LIN {X 0,Y 581.14,Z 534.428,A -85,B 0,C 180,E1 -1994.848,E2 -1994.848} C_VEL
LIN {X 0,Y 580.577,Z 528.636,A -85,B 0,C 180,E1 -1994.951,E2 -1994.951} C_VEL
LIN {X 0,Y 575.005,Z 509.982,A -85,B 0,C 180,E1 -1995.336,E2 -1995.336} C_VEL
LIN {X 0,Y 574.391,Z 504.171,A -85,B 0,C 180,E1 -1995.426,E2 -1995.426} C_VEL
LIN {X 0,Y 574.468,Z 402.044,A -85,B 0,C 180,E1 -1996.725,E2 -1996.725} C_VEL
LIN {X 0,Y 573.703,Z 397.536,A -85,B 0,C 180,E1 -1996.823,E2 -1996.823} C_VEL
LIN {X 0,Y 573.883,Z 376.717,A -85,B 0,C 180,E1 -1999.443,E2 -1999.443} C_VEL
LIN {X 0,Y 574.185,Z 354.585,A -85,B 0,C 180,E1 -2002.299,E2 -2002.299} C_VEL
LIN {X 0,Y 574.353,Z 340.111,A -85,B 0,C 180,E1 -2004.2,E2 -2004.2} C_VEL
LIN {X 0,Y 573.485,Z 334.982,A -85,B 0,C 180,E1 -2004.924,E2 -2004.924} C_VEL
LIN {X 0,Y 573.218,Z 333.802,A -85,B 0,C 180,E1 -2005.15,E2 -2005.15} C_VEL
LIN {X 0,Y 573.188,Z 333.715,A -85,B 0,C 180,E1 -2008.016,E2 -2008.016} C_VEL
LIN {X 0,Y 573.207,Z 333.705,A -85,B 0,C 180,E1 -2010.878,E2 -2010.878} C_VEL
LIN {X 0,Y 573.216,Z 333.705,A -85,B 0,C 180,E1 -2013.517,E2 -2013.517} C_VEL
LIN {X 0,Y 573.178,Z 333.717,A -85,B 0,C 180,E1 -2016.054,E2 -2016.054} C_VEL
LIN {X 0,Y 573.212,Z 333.704,A -85,B 0,C 180,E1 -2018.704,E2 -2018.704} C_VEL
LIN {X 0,Y 573.184,Z 333.709,A -85,B 0,C 180,E1 -2021.587,E2 -2021.587} C_VEL
LIN {X 0,Y 573.203,Z 333.71,A -85,B 0,C 180,E1 -2024.337,E2 -2024.337} C_VEL
LIN {X 0,Y 573.207,Z 333.702,A -85,B 0,C 180,E1 -2027.362,E2 -2027.362} C_VEL
LIN {X 0,Y 573.219,Z 333.704,A -85,B 0,C 180,E1 -2030.572,E2 -2030.572} C_VEL
LIN {X 0,Y 573.199,Z 333.703,A -85,B 0,C 180,E1 -2033.073,E2 -2033.073} C_VEL
LIN {X 0,Y 573.237,Z 333.704,A -85,B 0,C 180,E1 -2035.669,E2 -2035.669} C_VEL
LIN {X 0,Y 573.207,Z 333.713,A -85,B 0,C 180,E1 -2038.182,E2 -2038.182} C_VEL
LIN {X 0,Y 573.218,Z 333.707,A -85,B 0,C 180,E1 -2040.631,E2 -2040.631} C_VEL
LIN {X 0,Y 573.235,Z 333.849,A -85,B 0,C 180,E1 -2042.826,E2 -2042.826} C_VEL
LIN {X 0,Y 574.862,Z 341.006,A -85,B 0,C 180,E1 -2043.754,E2 -2043.754} C_VEL
LIN {X 0,Y 574.556,Z 361.798,A -85,B 0,C 180,E1 -2046.193,E2 -2046.193} C_VEL
LIN {X 0,Y 574.194,Z 387.884,A -85,B 0,C 180,E1 -2049.209,E2 -2049.209} C_VEL
LIN {X 0,Y 574.072,Z 398.599,A -85,B 0,C 180,E1 -2050.415,E2 -2050.415} C_VEL
LIN {X 0,Y 575.202,Z 405.826,A -85,B 0,C 180,E1 -2050.567,E2 -2050.567} C_VEL
LIN {X 0,Y 574.722,Z 563.783,A -85,B 0,C 180,E1 -2052.608,E2 -2052.608} C_VEL
LIN {X 0,Y 574.651,Z 578.295,A -85,B 0,C 180,E1 -2052.915,E2 -2052.915} C_VEL
LIN {X 0,Y 574.422,Z 594.793,A -85,B 0,C 180,E1 -2053.428,E2 -2053.428} C_VEL
LIN {X 0,Y 574.286,Z 608.726,A -85,B 0,C 180,E1 -2054.017,E2 -2054.017} C_VEL
LIN {X 0,Y 574.055,Z 620.862,A -85,B 0,C 180,E1 -2054.648,E2 -2054.648} C_VEL
LIN {X 0,Y 573.885,Z 634.297,A -85,B 0,C 180,E1 -2055.496,E2 -2055.496} C_VEL
LIN {X 0,Y 573.651,Z 647.761,A -85,B 0,C 180,E1 -2056.539,E2 -2056.539} C_VEL
LIN {X 0,Y 573.524,Z 657.489,A -85,B 0,C 180,E1 -2057.437,E2 -2057.437} C_VEL
LIN {X 0,Y 573.349,Z 667.502,A -85,B 0,C 180,E1 -2058.51,E2 -2058.51} C_VEL
LIN {X 0,Y 573.274,Z 677.322,A -85,B 0,C 180,E1 -2059.76,E2 -2059.76} C_VEL
LIN {X 0,Y 573.133,Z 686.46,A -85,B 0,C 180,E1 -2061.183,E2 -2061.183} C_VEL
LIN {X 0,Y 573.095,Z 692.191,A -85,B 0,C 180,E1 -2062.247,E2 -2062.247} C_VEL
LIN {X 0,Y 573.013,Z 698.405,A -85,B 0,C 180,E1 -2063.662,E2 -2063.662} C_VEL
LIN {X 0,Y 572.998,Z 702.164,A -85,B 0,C 180,E1 -2064.722,E2 -2064.722} C_VEL
LIN {X 0,Y 573.008,Z 705.165,A -85,B 0,C 180,E1 -2065.78,E2 -2065.78} C_VEL
LIN {X 0,Y 572.953,Z 708.114,A -85,B 0,C 180,E1 -2067.188,E2 -2067.188} C_VEL
LIN {X 0,Y 572.942,Z 709.884,A -85,B 0,C 180,E1 -2068.594,E2 -2068.594} C_VEL
LIN {X 0,Y 572.936,Z 710.496,A -85,B 0,C 180,E1 -2070,E2 -2070} C_VEL
LIN {X 0,Y 572.944,Z 709.958,A -85,B 0,C 180,E1 -2071.406,E2 -2071.406} C_VEL
LIN {X 0,Y 572.956,Z 708.262,A -85,B 0,C 180,E1 -2072.812,E2 -2072.812} C_VEL
LIN {X 0,Y 573.008,Z 705.388,A -85,B 0,C 180,E1 -2074.22,E2 -2074.22} C_VEL
LIN {X 0,Y 573.054,Z 701.325,A -85,B 0,C 180,E1 -2075.63,E2 -2075.63} C_VEL
LIN {X 0,Y 573.049,Z 695.916,A -85,B 0,C 180,E1 -2077.045,E2 -2077.045} C_VEL
LIN {X 0,Y 573.099,Z 688.976,A -85,B 0,C 180,E1 -2078.462,E2 -2078.462} C_VEL
LIN {X 0,Y 573.188,Z 681.545,A -85,B 0,C 180,E1 -2079.706,E2 -2079.706} C_VEL
LIN {X 0,Y 573.287,Z 673.107,A -85,B 0,C 180,E1 -2080.89,E2 -2080.89} C_VEL
LIN {X 0,Y 573.406,Z 663.566,A -85,B 0,C 180,E1 -2082.026,E2 -2082.026} C_VEL
LIN {X 0,Y 573.609,Z 651.863,A -85,B 0,C 180,E1 -2083.191,E2 -2083.191} C_VEL
LIN {X 0,Y 573.777,Z 639.91,A -85,B 0,C 180,E1 -2084.18,E2 -2084.18} C_VEL
LIN {X 0,Y 574.002,Z 628.328,A -85,B 0,C 180,E1 -2084.99,E2 -2084.99} C_VEL
LIN {X 0,Y 574.168,Z 616.021,A -85,B 0,C 180,E1 -2085.713,E2 -2085.713} C_VEL
LIN {X 0,Y 574.347,Z 600.523,A -85,B 0,C 180,E1 -2086.437,E2 -2086.437} C_VEL
LIN {X 0,Y 574.505,Z 586.676,A -85,B 0,C 180,E1 -2086.936,E2 -2086.936} C_VEL
LIN {X 0,Y 574.677,Z 572.66,A -85,B 0,C 180,E1 -2087.311,E2 -2087.311} C_VEL
LIN {X 0,Y 574.793,Z 556.718,A -85,B 0,C 180,E1 -2087.589,E2 -2087.589} C_VEL
LIN {X 0,Y 575.167,Z 404.401,A -85,B 0,C 180,E1 -2089.542,E2 -2089.542} C_VEL
LIN {X 0,Y 574.062,Z 398.56,A -85,B 0,C 180,E1 -2089.678,E2 -2089.678} C_VEL
LIN {X 0,Y 574.415,Z 372.355,A -85,B 0,C 180,E1 -2092.669,E2 -2092.669} C_VEL
LIN {X 0,Y 574.801,Z 346.251,A -85,B 0,C 180,E1 -2095.725,E2 -2095.725} C_VEL
LIN {X 0,Y 574.791,Z 340.48,A -85,B 0,C 180,E1 -2096.4,E2 -2096.4} C_VEL
LIN {X 0,Y 573.231,Z 333.822,A -85,B 0,C 180,E1 -2097.273,E2 -2097.273} C_VEL
LIN {X 0,Y 573.219,Z 333.71,A -85,B 0,C 180,E1 -2100.178,E2 -2100.178} C_VEL
LIN {X 0,Y 573.216,Z 333.704,A -85,B 0,C 180,E1 -2102.647,E2 -2102.647} C_VEL
LIN {X 0,Y 573.178,Z 333.709,A -85,B 0,C 180,E1 -2105.19,E2 -2105.19} C_VEL
LIN {X 0,Y 573.207,Z 333.712,A -85,B 0,C 180,E1 -2107.81,E2 -2107.81} C_VEL
LIN {X 0,Y 573.199,Z 333.706,A -85,B 0,C 180,E1 -2110.529,E2 -2110.529} C_VEL
LIN {X 0,Y 573.193,Z 333.707,A -85,B 0,C 180,E1 -2113.363,E2 -2113.363} C_VEL
LIN {X 0,Y 573.217,Z 333.709,A -85,B 0,C 180,E1 -2115.665,E2 -2115.665} C_VEL
LIN {X 0,Y 573.191,Z 333.707,A -85,B 0,C 180,E1 -2118.539,E2 -2118.539} C_VEL
LIN {X 0,Y 573.229,Z 333.703,A -85,B 0,C 180,E1 -2121.297,E2 -2121.297} C_VEL
LIN {X 0,Y 573.184,Z 333.711,A -85,B 0,C 180,E1 -2124.023,E2 -2124.023} C_VEL
LIN {X 0,Y 573.231,Z 333.701,A -85,B 0,C 180,E1 -2126.515,E2 -2126.515} C_VEL
LIN {X 0,Y 573.224,Z 333.701,A -85,B 0,C 180,E1 -2129.119,E2 -2129.119} C_VEL
LIN {X 0,Y 573.219,Z 333.705,A -85,B 0,C 180,E1 -2131.977,E2 -2131.977} C_VEL
LIN {X 0,Y 573.223,Z 333.701,A -85,B 0,C 180,E1 -2134.588,E2 -2134.588} C_VEL
LIN {X 0,Y 573.236,Z 333.7,A -85,B 0,C 180,E1 -2136.901,E2 -2136.901} C_VEL
LIN {X 0,Y 573.249,Z 333.7,A -85,B 0,C 180,E1 -2139.173,E2 -2139.173} C_VEL
LIN {X 0,Y 573.21,Z 333.71,A -85,B 0,C 180,E1 -2141.411,E2 -2141.411} C_VEL
LIN {X 0,Y 573.238,Z 333.707,A -85,B 0,C 180,E1 -2143.621,E2 -2143.621} C_VEL
LIN {X 0,Y 573.272,Z 333.701,A -85,B 0,C 180,E1 -2145.807,E2 -2145.807} C_VEL
LIN {X 0,Y 573.265,Z 333.694,A -85,B 0,C 180,E1 -2148.745,E2 -2148.745} C_VEL
LIN {X 0,Y 573.281,Z 333.704,A -85,B 0,C 180,E1 -2151.54,E2 -2151.54} C_VEL
LIN {X 0,Y 573.244,Z 333.704,A -85,B 0,C 180,E1 -2153.665,E2 -2153.665} C_VEL
LIN {X 0,Y 573.228,Z 333.704,A -85,B 0,C 180,E1 -2155.781,E2 -2155.781} C_VEL
LIN {X 0,Y 573.314,Z 333.693,A -85,B 0,C 180,E1 -2157.892,E2 -2157.892} C_VEL
LIN {X 0,Y 573.32,Z 333.689,A -85,B 0,C 180,E1 -2160.702,E2 -2160.702} C_VEL
LIN {X 0,Y 573.294,Z 333.692,A -85,B 0,C 180,E1 -2162.811,E2 -2162.811} C_VEL
LIN {X 0,Y 573.295,Z 333.697,A -85,B 0,C 180,E1 -2165.628,E2 -2165.628} C_VEL
LIN {X 0,Y 573.255,Z 333.695,A -85,B 0,C 180,E1 -2168.46,E2 -2168.46} C_VEL
LIN {X 0,Y 573.274,Z 333.704,A -85,B 0,C 180,E1 -2171.312,E2 -2171.312} C_VEL
LIN {X 0,Y 573.261,Z 333.694,A -85,B 0,C 180,E1 -2174.193,E2 -2174.193} C_VEL
LIN {X 0,Y 573.259,Z 333.704,A -85,B 0,C 180,E1 -2177.111,E2 -2177.111} C_VEL
LIN {X 0,Y 573.241,Z 333.697,A -85,B 0,C 180,E1 -2180.077,E2 -2180.077} C_VEL
LIN {X 0,Y 573.235,Z 333.7,A -85,B 0,C 180,E1 -2182.338,E2 -2182.338} C_VEL
LIN {X 0,Y 573.254,Z 333.703,A -85,B 0,C 180,E1 -2185.41,E2 -2185.41} C_VEL
LIN {X 0,Y 573.25,Z 333.698,A -85,B 0,C 180,E1 -2188.029,E2 -2188.029} C_VEL
LIN {X 0,Y 573.234,Z 333.704,A -85,B 0,C 180,E1 -2190.883,E2 -2190.883} C_VEL
LIN {X 0,Y 573.263,Z 333.698,A -85,B 0,C 180,E1 -2193.524,E2 -2193.524} C_VEL
LIN {X 0,Y 573.215,Z 333.702,A -85,B 0,C 180,E1 -2196.051,E2 -2196.051} C_VEL
LIN {X 0,Y 573.25,Z 333.701,A -85,B 0,C 180,E1 -2198.701,E2 -2198.701} C_VEL
LIN {X 0,Y 573.244,Z 333.699,A -85,B 0,C 180,E1 -2201.594,E2 -2201.594} C_VEL
LIN {X 0,Y 573.236,Z 333.701,A -85,B 0,C 180,E1 -2204.333,E2 -2204.333} C_VEL
LIN {X 0,Y 573.24,Z 333.702,A -85,B 0,C 180,E1 -2207.358,E2 -2207.358} C_VEL
LIN {X 0,Y 573.248,Z 333.701,A -85,B 0,C 180,E1 -2210.393,E2 -2210.393} C_VEL
LIN {X 0,Y 573.253,Z 333.705,A -85,B 0,C 180,E1 -2213.078,E2 -2213.078} C_VEL
LIN {X 0,Y 573.266,Z 333.697,A -85,B 0,C 180,E1 -2215.671,E2 -2215.671} C_VEL
LIN {X 0,Y 573.247,Z 333.7,A -85,B 0,C 180,E1 -2218.185,E2 -2218.185} C_VEL
LIN {X 0,Y 573.264,Z 333.704,A -85,B 0,C 180,E1 -2220.634,E2 -2220.634} C_VEL
LIN {X 0,Y 573.273,Z 333.826,A -85,B 0,C 180,E1 -2223.522,E2 -2223.522} C_VEL
LIN {X 0,Y 574.8,Z 339.819,A -85,B 0,C 180,E1 -2224.275,E2 -2224.275} C_VEL
LIN {X 0,Y 574.832,Z 350.617,A -85,B 0,C 180,E1 -2225.437,E2 -2225.437} C_VEL
LIN {X 0,Y 574.354,Z 379.411,A -85,B 0,C 180,E1 -2228.464,E2 -2228.464} C_VEL
LIN {X 0,Y 574.163,Z 397.928,A -85,B 0,C 180,E1 -2230.363,E2 -2230.363} C_VEL
LIN {X 0,Y 575.245,Z 404.725,A -85,B 0,C 180,E1 -2230.51,E2 -2230.51} C_VEL
LIN {X 0,Y 574.744,Z 565.38,A -85,B 0,C 180,E1 -2232.586,E2 -2232.586} C_VEL
LIN {X 0,Y 574.616,Z 580.708,A -85,B 0,C 180,E1 -2232.93,E2 -2232.93} C_VEL
LIN {X 0,Y 574.433,Z 596.043,A -85,B 0,C 180,E1 -2233.428,E2 -2233.428} C_VEL
LIN {X 0,Y 574.292,Z 609.771,A -85,B 0,C 180,E1 -2234.017,E2 -2234.017} C_VEL
LIN {X 0,Y 574.032,Z 623.244,A -85,B 0,C 180,E1 -2234.738,E2 -2234.738} C_VEL
LIN {X 0,Y 573.861,Z 636.818,A -85,B 0,C 180,E1 -2235.632,E2 -2235.632} C_VEL
LIN {X 0,Y 573.635,Z 649.35,A -85,B 0,C 180,E1 -2236.629,E2 -2236.629} C_VEL
LIN {X 0,Y 573.477,Z 659.749,A -85,B 0,C 180,E1 -2237.616,E2 -2237.616} C_VEL
LIN {X 0,Y 573.286,Z 669.77,A -85,B 0,C 180,E1 -2238.734,E2 -2238.734} C_VEL
LIN {X 0,Y 573.243,Z 678.858,A -85,B 0,C 180,E1 -2239.939,E2 -2239.939} C_VEL
LIN {X 0,Y 573.132,Z 686.734,A -85,B 0,C 180,E1 -2241.183,E2 -2241.183} C_VEL
LIN {X 0,Y 573.074,Z 694.089,A -85,B 0,C 180,E1 -2242.602,E2 -2242.602} C_VEL
LIN {X 0,Y 573.041,Z 699.923,A -85,B 0,C 180,E1 -2244.016,E2 -2244.016} C_VEL
LIN {X 0,Y 572.951,Z 703.385,A -85,B 0,C 180,E1 -2245.074,E2 -2245.074} C_VEL
LIN {X 0,Y 573.005,Z 706.889,A -85,B 0,C 180,E1 -2246.484,E2 -2246.484} C_VEL
LIN {X 0,Y 572.938,Z 709.192,A -85,B 0,C 180,E1 -2247.891,E2 -2247.891} C_VEL
LIN {X 0,Y 572.936,Z 710.349,A -85,B 0,C 180,E1 -2249.297,E2 -2249.297} C_VEL
LIN {X 0,Y 572.936,Z 710.349,A -85,B 0,C 180,E1 -2250.703,E2 -2250.703} C_VEL
LIN {X 0,Y 572.938,Z 709.191,A -85,B 0,C 180,E1 -2252.109,E2 -2252.109} C_VEL
LIN {X 0,Y 573.005,Z 706.887,A -85,B 0,C 180,E1 -2253.516,E2 -2253.516} C_VEL
LIN {X 0,Y 572.951,Z 703.385,A -85,B 0,C 180,E1 -2254.926,E2 -2254.926} C_VEL
LIN {X 0,Y 573.013,Z 698.608,A -85,B 0,C 180,E1 -2256.338,E2 -2256.338} C_VEL
LIN {X 0,Y 573.094,Z 692.422,A -85,B 0,C 180,E1 -2257.753,E2 -2257.753} C_VEL
LIN {X 0,Y 573.135,Z 684.648,A -85,B 0,C 180,E1 -2259.173,E2 -2259.173} C_VEL
LIN {X 0,Y 573.27,Z 676.368,A -85,B 0,C 180,E1 -2260.418,E2 -2260.418} C_VEL
LIN {X 0,Y 573.386,Z 666.39,A -85,B 0,C 180,E1 -2261.668,E2 -2261.668} C_VEL
LIN {X 0,Y 573.568,Z 656.188,A -85,B 0,C 180,E1 -2262.742,E2 -2262.742} C_VEL
LIN {X 0,Y 573.705,Z 644.017,A -85,B 0,C 180,E1 -2263.82,E2 -2263.82} C_VEL
LIN {X 0,Y 573.962,Z 630.901,A -85,B 0,C 180,E1 -2264.781,E2 -2264.781} C_VEL
LIN {X 0,Y 574.141,Z 616.867,A -85,B 0,C 180,E1 -2265.623,E2 -2265.623} C_VEL
LIN {X 0,Y 574.351,Z 602.795,A -85,B 0,C 180,E1 -2266.3,E2 -2266.3} C_VEL
LIN {X 0,Y 574.526,Z 588.3,A -85,B 0,C 180,E1 -2266.844,E2 -2266.844} C_VEL
LIN {X 0,Y 574.714,Z 572.326,A -85,B 0,C 180,E1 -2267.276,E2 -2267.276} C_VEL
LIN {X 0,Y 574.804,Z 556.362,A -85,B 0,C 180,E1 -2267.548,E2 -2267.548} C_VEL
LIN {X 0,Y 575.079,Z 403.047,A -85,B 0,C 180,E1 -2269.518,E2 -2269.518} C_VEL
LIN {X 0,Y 574.164,Z 397.918,A -85,B 0,C 180,E1 -2269.637,E2 -2269.637} C_VEL
LIN {X 0,Y 574.502,Z 370.411,A -85,B 0,C 180,E1 -2272.476,E2 -2272.476} C_VEL
LIN {X 0,Y 574.942,Z 343.417,A -85,B 0,C 180,E1 -2275.33,E2 -2275.33} C_VEL
LIN {X 0,Y 574.8,Z 339.818,A -85,B 0,C 180,E1 -2275.725,E2 -2275.725} C_VEL
LIN {X 0,Y 573.272,Z 333.818,A -85,B 0,C 180,E1 -2276.477,E2 -2276.477} C_VEL
LIN {X 0,Y 573.265,Z 333.704,A -85,B 0,C 180,E1 -2279.366,E2 -2279.366} C_VEL
LIN {X 0,Y 573.251,Z 333.7,A -85,B 0,C 180,E1 -2282.228,E2 -2282.228} C_VEL
LIN {X 0,Y 573.242,Z 333.708,A -85,B 0,C 180,E1 -2284.772,E2 -2284.772} C_VEL
LIN {X 0,Y 573.237,Z 333.701,A -85,B 0,C 180,E1 -2287.808,E2 -2287.808} C_VEL
LIN {X 0,Y 573.246,Z 333.706,A -85,B 0,C 180,E1 -2290.525,E2 -2290.525} C_VEL
LIN {X 0,Y 573.232,Z 333.702,A -85,B 0,C 180,E1 -2293.36,E2 -2293.36} C_VEL
LIN {X 0,Y 573.237,Z 333.706,A -85,B 0,C 180,E1 -2296.332,E2 -2296.332} C_VEL
LIN {X 0,Y 573.227,Z 333.711,A -85,B 0,C 180,E1 -2298.543,E2 -2298.543} C_VEL
LIN {X 0,Y 573.236,Z 333.701,A -85,B 0,C 180,E1 -2301.298,E2 -2301.298} C_VEL
LIN {X 0,Y 573.188,Z 333.711,A -85,B 0,C 180,E1 -2304.022,E2 -2304.022} C_VEL
LIN {X 0,Y 573.252,Z 333.706,A -85,B 0,C 180,E1 -2306.517,E2 -2306.517} C_VEL
LIN {X 0,Y 573.219,Z 333.704,A -85,B 0,C 180,E1 -2309.12,E2 -2309.12} C_VEL
LIN {X 0,Y 573.193,Z 333.714,A -85,B 0,C 180,E1 -2311.983,E2 -2311.983} C_VEL
LIN {X 0,Y 573.215,Z 333.77,A -85,B 0,C 180,E1 -2314.897,E2 -2314.897} C_VEL
LIN {X 0,Y 573.372,Z 334.597,A -85,B 0,C 180,E1 -2315.1,E2 -2315.1} C_VEL
LIN {X 0,Y 574.37,Z 339.464,A -85,B 0,C 180,E1 -2315.801,E2 -2315.801} C_VEL
LIN {X 0,Y 574.135,Z 356.794,A -85,B 0,C 180,E1 -2318.078,E2 -2318.078} C_VEL
LIN {X 0,Y 573.873,Z 376.043,A -85,B 0,C 180,E1 -2320.56,E2 -2320.56} C_VEL
LIN {X 0,Y 573.692,Z 397.29,A -85,B 0,C 180,E1 -2323.246,E2 -2323.246} C_VEL
LIN {X 0,Y 574.133,Z 400.139,A -85,B 0,C 180,E1 -2323.331,E2 -2323.331} C_VEL
LIN {X 0,Y 574.604,Z 403.469,A -85,B 0,C 180,E1 -2323.387,E2 -2323.387} C_VEL
LIN {X 0,Y 574.282,Z 535.959,A -85,B 0,C 180,E1 -2325.086,E2 -2325.086} C_VEL
LIN {X 0,Y 574.173,Z 550.401,A -85,B 0,C 180,E1 -2325.421,E2 -2325.421} C_VEL
LIN {X 0,Y 574.032,Z 564.86,A -85,B 0,C 180,E1 -2325.917,E2 -2325.917} C_VEL
LIN {X 0,Y 573.847,Z 578.493,A -85,B 0,C 180,E1 -2326.544,E2 -2326.544} C_VEL
LIN {X 0,Y 573.713,Z 590.81,A -85,B 0,C 180,E1 -2327.262,E2 -2327.262} C_VEL
LIN {X 0,Y 573.535,Z 602.03,A -85,B 0,C 180,E1 -2328.066,E2 -2328.066} C_VEL
LIN {X 0,Y 573.438,Z 613.674,A -85,B 0,C 180,E1 -2329.081,E2 -2329.081} C_VEL
LIN {X 0,Y 573.242,Z 623.482,A -85,B 0,C 180,E1 -2330.117,E2 -2330.117} C_VEL
LIN {X 0,Y 573.202,Z 631.851,A -85,B 0,C 180,E1 -2331.184,E2 -2331.184} C_VEL
LIN {X 0,Y 573.111,Z 639.88,A -85,B 0,C 180,E1 -2332.425,E2 -2332.425} C_VEL
LIN {X 0,Y 573.021,Z 646.33,A -85,B 0,C 180,E1 -2333.663,E2 -2333.663} C_VEL
LIN {X 0,Y 573,Z 650.771,A -85,B 0,C 180,E1 -2334.722,E2 -2334.722} C_VEL
LIN {X 0,Y 573.029,Z 654.297,A -85,B 0,C 180,E1 -2335.78,E2 -2335.78} C_VEL
LIN {X 0,Y 572.957,Z 657.752,A -85,B 0,C 180,E1 -2337.188,E2 -2337.188} C_VEL
LIN {X 0,Y 572.944,Z 659.767,A -85,B 0,C 180,E1 -2338.594,E2 -2338.594} C_VEL
LIN {X 0,Y 572.937,Z 660.496,A -85,B 0,C 180,E1 -2340,E2 -2340} C_VEL
LIN {X 0,Y 572.941,Z 659.852,A -85,B 0,C 180,E1 -2341.406,E2 -2341.406} C_VEL
LIN {X 0,Y 572.954,Z 657.929,A -85,B 0,C 180,E1 -2342.812,E2 -2342.812} C_VEL
LIN {X 0,Y 573.029,Z 654.565,A -85,B 0,C 180,E1 -2344.22,E2 -2344.22} C_VEL
LIN {X 0,Y 573.057,Z 649.763,A -85,B 0,C 180,E1 -2345.631,E2 -2345.631} C_VEL
LIN {X 0,Y 573.066,Z 645.029,A -85,B 0,C 180,E1 -2346.699,E2 -2346.699} C_VEL
LIN {X 0,Y 573.117,Z 638.313,A -85,B 0,C 180,E1 -2347.93,E2 -2347.93} C_VEL
LIN {X 0,Y 573.22,Z 629.885,A -85,B 0,C 180,E1 -2349.171,E2 -2349.171} C_VEL
LIN {X 0,Y 573.304,Z 621.136,A -85,B 0,C 180,E1 -2350.239,E2 -2350.239} C_VEL
LIN {X 0,Y 573.463,Z 610.478,A -85,B 0,C 180,E1 -2351.308,E2 -2351.308} C_VEL
LIN {X 0,Y 573.613,Z 599.736,A -85,B 0,C 180,E1 -2352.202,E2 -2352.202} C_VEL
LIN {X 0,Y 573.758,Z 587.972,A -85,B 0,C 180,E1 -2353.007,E2 -2353.007} C_VEL
LIN {X 0,Y 573.936,Z 575.01,A -85,B 0,C 180,E1 -2353.724,E2 -2353.724} C_VEL
LIN {X 0,Y 574.086,Z 561.993,A -85,B 0,C 180,E1 -2354.285,E2 -2354.285} C_VEL
LIN {X 0,Y 574.194,Z 547.655,A -85,B 0,C 180,E1 -2354.743,E2 -2354.743} C_VEL
LIN {X 0,Y 574.311,Z 533.037,A -85,B 0,C 180,E1 -2355.05,E2 -2355.05} C_VEL
LIN {X 0,Y 574.391,Z 504.171,A -85,B 0,C 180,E1 -2355.426,E2 -2355.426} C_VEL
LIN {X 0,Y 573.789,Z 498.365,A -85,B 0,C 180,E1 -2355.516,E2 -2355.516} C_VEL
LIN {X 0,Y 568.261,Z 479.712,A -85,B 0,C 180,E1 -2355.91,E2 -2355.91} C_VEL
LIN {X 0,Y 567.626,Z 473.907,A -85,B 0,C 180,E1 -2356.003,E2 -2356.003} C_VEL
LIN {X 0,Y 567.759,Z 403.527,A -85,B 0,C 180,E1 -2356.909,E2 -2356.909} C_VEL
LIN {X 0,Y 566.721,Z 397.449,A -85,B 0,C 180,E1 -2357.041,E2 -2357.041} C_VEL
LIN {X 0,Y 566.977,Z 376.456,A -85,B 0,C 180,E1 -2359.723,E2 -2359.723} C_VEL
LIN {X 0,Y 567.365,Z 353.15,A -85,B 0,C 180,E1 -2362.774,E2 -2362.774} C_VEL
LIN {X 0,Y 567.523,Z 341.61,A -85,B 0,C 180,E1 -2364.315,E2 -2364.315} C_VEL
LIN {X 0,Y 566.207,Z 334.732,A -85,B 0,C 180,E1 -2365.336,E2 -2365.336} C_VEL
LIN {X 0,Y 566.133,Z 334.594,A -85,B 0,C 180,E1 -2368.188,E2 -2368.188} C_VEL
LIN {X 0,Y 566.172,Z 334.581,A -85,B 0,C 180,E1 -2371.073,E2 -2371.073} C_VEL
LIN {X 0,Y 566.179,Z 334.585,A -85,B 0,C 180,E1 -2373.729,E2 -2373.729} C_VEL
LIN {X 0,Y 566.13,Z 334.588,A -85,B 0,C 180,E1 -2376.575,E2 -2376.575} C_VEL
LIN {X 0,Y 566.193,Z 334.578,A -85,B 0,C 180,E1 -2379.276,E2 -2379.276} C_VEL
LIN {X 0,Y 566.141,Z 334.589,A -85,B 0,C 180,E1 -2382.094,E2 -2382.094} C_VEL
LIN {X 0,Y 566.154,Z 334.582,A -85,B 0,C 180,E1 -2385.038,E2 -2385.038} C_VEL
LIN {X 0,Y 566.135,Z 334.594,A -85,B 0,C 180,E1 -2388.146,E2 -2388.146} C_VEL
LIN {X 0,Y 566.191,Z 334.578,A -85,B 0,C 180,E1 -2390.724,E2 -2390.724} C_VEL
LIN {X 0,Y 566.13,Z 334.586,A -85,B 0,C 180,E1 -2393.425,E2 -2393.425} C_VEL
LIN {X 0,Y 566.178,Z 334.587,A -85,B 0,C 180,E1 -2396.271,E2 -2396.271} C_VEL
LIN {X 0,Y 566.173,Z 334.581,A -85,B 0,C 180,E1 -2398.927,E2 -2398.927} C_VEL
LIN {X 0,Y 566.134,Z 334.593,A -85,B 0,C 180,E1 -2401.853,E2 -2401.853} C_VEL
LIN {X 0,Y 566.202,Z 334.799,A -85,B 0,C 180,E1 -2402.635,E2 -2402.635} C_VEL
LIN {X 0,Y 567.919,Z 341.773,A -85,B 0,C 180,E1 -2403.545,E2 -2403.545} C_VEL
LIN {X 0,Y 567.826,Z 356.843,A -85,B 0,C 180,E1 -2405.309,E2 -2405.309} C_VEL
LIN {X 0,Y 567.412,Z 379.738,A -85,B 0,C 180,E1 -2407.995,E2 -2407.995} C_VEL
LIN {X 0,Y 567.174,Z 398.798,A -85,B 0,C 180,E1 -2410.177,E2 -2410.177} C_VEL
LIN {X 0,Y 568.513,Z 406.202,A -85,B 0,C 180,E1 -2410.334,E2 -2410.334} C_VEL
LIN {X 0,Y 567.958,Z 563.751,A -85,B 0,C 180,E1 -2412.394,E2 -2412.394} C_VEL
LIN {X 0,Y 567.867,Z 577.741,A -85,B 0,C 180,E1 -2412.69,E2 -2412.69} C_VEL
LIN {X 0,Y 567.638,Z 593.61,A -85,B 0,C 180,E1 -2413.177,E2 -2413.177} C_VEL
LIN {X 0,Y 567.462,Z 606.818,A -85,B 0,C 180,E1 -2413.727,E2 -2413.727} C_VEL
LIN {X 0,Y 567.251,Z 619.256,A -85,B 0,C 180,E1 -2414.367,E2 -2414.367} C_VEL
LIN {X 0,Y 567.033,Z 630.566,A -85,B 0,C 180,E1 -2415.063,E2 -2415.063} C_VEL
LIN {X 0,Y 566.795,Z 642.267,A -85,B 0,C 180,E1 -2415.916,E2 -2415.916} C_VEL
LIN {X 0,Y 566.572,Z 653.824,A -85,B 0,C 180,E1 -2416.916,E2 -2416.916} C_VEL
LIN {X 0,Y 566.401,Z 664.383,A -85,B 0,C 180,E1 -2418.004,E2 -2418.004} C_VEL
LIN {X 0,Y 566.263,Z 672.95,A -85,B 0,C 180,E1 -2419.044,E2 -2419.044} C_VEL
LIN {X 0,Y 566.13,Z 680.949,A -85,B 0,C 180,E1 -2420.172,E2 -2420.172} C_VEL
LIN {X 0,Y 566.064,Z 688.465,A -85,B 0,C 180,E1 -2421.432,E2 -2421.432} C_VEL
LIN {X 0,Y 565.975,Z 695.51,A -85,B 0,C 180,E1 -2422.867,E2 -2422.867} C_VEL
LIN {X 0,Y 565.981,Z 701.025,A -85,B 0,C 180,E1 -2424.299,E2 -2424.299} C_VEL
LIN {X 0,Y 565.913,Z 705.162,A -85,B 0,C 180,E1 -2425.727,E2 -2425.727} C_VEL
LIN {X 0,Y 565.872,Z 708.108,A -85,B 0,C 180,E1 -2427.152,E2 -2427.152} C_VEL
LIN {X 0,Y 565.842,Z 709.879,A -85,B 0,C 180,E1 -2428.576,E2 -2428.576} C_VEL
LIN {X 0,Y 565.837,Z 710.496,A -85,B 0,C 180,E1 -2430,E2 -2430} C_VEL
LIN {X 0,Y 565.843,Z 709.96,A -85,B 0,C 180,E1 -2431.423,E2 -2431.423} C_VEL
LIN {X 0,Y 565.874,Z 708.262,A -85,B 0,C 180,E1 -2432.847,E2 -2432.847} C_VEL
LIN {X 0,Y 565.913,Z 705.381,A -85,B 0,C 180,E1 -2434.273,E2 -2434.273} C_VEL
LIN {X 0,Y 565.981,Z 701.316,A -85,B 0,C 180,E1 -2435.701,E2 -2435.701} C_VEL
LIN {X 0,Y 565.974,Z 695.914,A -85,B 0,C 180,E1 -2437.133,E2 -2437.133} C_VEL
LIN {X 0,Y 566.047,Z 688.967,A -85,B 0,C 180,E1 -2438.568,E2 -2438.568} C_VEL
LIN {X 0,Y 566.125,Z 681.533,A -85,B 0,C 180,E1 -2439.828,E2 -2439.828} C_VEL
LIN {X 0,Y 566.253,Z 673.626,A -85,B 0,C 180,E1 -2440.956,E2 -2440.956} C_VEL
LIN {X 0,Y 566.415,Z 663.564,A -85,B 0,C 180,E1 -2442.177,E2 -2442.177} C_VEL
LIN {X 0,Y 566.623,Z 651.845,A -85,B 0,C 180,E1 -2443.357,E2 -2443.357} C_VEL
LIN {X 0,Y 566.805,Z 641.073,A -85,B 0,C 180,E1 -2444.267,E2 -2444.267} C_VEL
LIN {X 0,Y 567.059,Z 629.676,A -85,B 0,C 180,E1 -2445.086,E2 -2445.086} C_VEL
LIN {X 0,Y 567.26,Z 617.619,A -85,B 0,C 180,E1 -2445.817,E2 -2445.817} C_VEL
LIN {X 0,Y 567.505,Z 602.75,A -85,B 0,C 180,E1 -2446.549,E2 -2446.549} C_VEL
LIN {X 0,Y 567.72,Z 588.08,A -85,B 0,C 180,E1 -2447.098,E2 -2447.098} C_VEL
LIN {X 0,Y 567.852,Z 575.243,A -85,B 0,C 180,E1 -2447.461,E2 -2447.461} C_VEL
LIN {X 0,Y 568.003,Z 561.651,A -85,B 0,C 180,E1 -2447.73,E2 -2447.73} C_VEL
LIN {X 0,Y 568.468,Z 405.474,A -85,B 0,C 180,E1 -2449.767,E2 -2449.767} C_VEL
LIN {X 0,Y 567.174,Z 398.477,A -85,B 0,C 180,E1 -2449.932,E2 -2449.932} C_VEL
LIN {X 0,Y 567.557,Z 373.981,A -85,B 0,C 180,E1 -2452.766,E2 -2452.766} C_VEL
LIN {X 0,Y 567.939,Z 350.401,A -85,B 0,C 180,E1 -2455.531,E2 -2455.531} C_VEL
LIN {X 0,Y 567.983,Z 342.532,A -85,B 0,C 180,E1 -2456.452,E2 -2456.452} C_VEL
LIN {X 0,Y 566.174,Z 334.674,A -85,B 0,C 180,E1 -2457.491,E2 -2457.491} C_VEL
LIN {X 0,Y 566.157,Z 334.585,A -85,B 0,C 180,E1 -2460.594,E2 -2460.594} C_VEL
LIN {X 0,Y 566.159,Z 334.582,A -85,B 0,C 180,E1 -2463.106,E2 -2463.106} C_VEL
LIN {X 0,Y 566.133,Z 334.592,A -85,B 0,C 180,E1 -2465.694,E2 -2465.694} C_VEL
LIN {X 0,Y 566.186,Z 334.579,A -85,B 0,C 180,E1 -2468.555,E2 -2468.555} C_VEL
LIN {X 0,Y 566.134,Z 334.585,A -85,B 0,C 180,E1 -2471.143,E2 -2471.143} C_VEL
LIN {X 0,Y 566.156,Z 334.588,A -85,B 0,C 180,E1 -2474.04,E2 -2474.04} C_VEL
LIN {X 0,Y 566.152,Z 334.584,A -85,B 0,C 180,E1 -2477.088,E2 -2477.088} C_VEL
LIN {X 0,Y 566.186,Z 334.58,A -85,B 0,C 180,E1 -2480.318,E2 -2480.318} C_VEL
LIN {X 0,Y 566.185,Z 334.579,A -85,B 0,C 180,E1 -2482.601,E2 -2482.601} C_VEL
LIN {X 0,Y 566.18,Z 334.579,A -85,B 0,C 180,E1 -2485.18,E2 -2485.18} C_VEL
LIN {X 0,Y 566.228,Z 334.58,A -85,B 0,C 180,E1 -2487.743,E2 -2487.743} C_VEL
LIN {X 0,Y 566.193,Z 334.579,A -85,B 0,C 180,E1 -2490.33,E2 -2490.33} C_VEL
LIN {X 0,Y 566.164,Z 334.578,A -85,B 0,C 180,E1 -2492.658,E2 -2492.658} C_VEL
LIN {X 0,Y 566.194,Z 334.578,A -85,B 0,C 180,E1 -2495.037,E2 -2495.037} C_VEL
LIN {X 0,Y 566.191,Z 334.578,A -85,B 0,C 180,E1 -2498.137,E2 -2498.137} C_VEL
LIN {X 0,Y 566.231,Z 334.572,A -85,B 0,C 180,E1 -2500.614,E2 -2500.614} C_VEL
LIN {X 0,Y 566.2,Z 334.581,A -85,B 0,C 180,E1 -2503.412,E2 -2503.412} C_VEL
LIN {X 0,Y 566.19,Z 334.578,A -85,B 0,C 180,E1 -2506.359,E2 -2506.359} C_VEL
LIN {X 0,Y 566.236,Z 334.569,A -85,B 0,C 180,E1 -2508.675,E2 -2508.675} C_VEL
LIN {X 0,Y 566.224,Z 334.581,A -85,B 0,C 180,E1 -2511.434,E2 -2511.434} C_VEL
LIN {X 0,Y 566.248,Z 334.568,A -85,B 0,C 180,E1 -2514.302,E2 -2514.302} C_VEL
LIN {X 0,Y 566.284,Z 334.569,A -85,B 0,C 180,E1 -2517.866,E2 -2517.866} C_VEL
LIN {X 0,Y 566.292,Z 334.564,A -85,B 0,C 180,E1 -2520.711,E2 -2520.711} C_VEL
LIN {X 0,Y 566.262,Z 334.568,A -85,B 0,C 180,E1 -2522.846,E2 -2522.846} C_VEL
LIN {X 0,Y 566.262,Z 334.572,A -85,B 0,C 180,E1 -2525.698,E2 -2525.698} C_VEL
LIN {X 0,Y 566.206,Z 334.573,A -85,B 0,C 180,E1 -2528.566,E2 -2528.566} C_VEL
LIN {X 0,Y 566.244,Z 334.577,A -85,B 0,C 180,E1 -2531.454,E2 -2531.454} C_VEL
LIN {X 0,Y 566.224,Z 334.571,A -85,B 0,C 180,E1 -2534.502,E2 -2534.502} C_VEL
LIN {X 0,Y 566.2,Z 334.584,A -85,B 0,C 180,E1 -2537.332,E2 -2537.332} C_VEL
LIN {X 0,Y 566.207,Z 334.573,A -85,B 0,C 180,E1 -2540.337,E2 -2540.337} C_VEL
LIN {X 0,Y 566.171,Z 334.587,A -85,B 0,C 180,E1 -2543.281,E2 -2543.281} C_VEL
LIN {X 0,Y 566.213,Z 334.576,A -85,B 0,C 180,E1 -2545.749,E2 -2545.749} C_VEL
LIN {X 0,Y 566.203,Z 334.576,A -85,B 0,C 180,E1 -2548.202,E2 -2548.202} C_VEL
LIN {X 0,Y 566.195,Z 334.584,A -85,B 0,C 180,E1 -2551.077,E2 -2551.077} C_VEL
LIN {X 0,Y 566.212,Z 334.574,A -85,B 0,C 180,E1 -2553.734,E2 -2553.734} C_VEL
LIN {X 0,Y 566.2,Z 334.579,A -85,B 0,C 180,E1 -2556.57,E2 -2556.57} C_VEL
LIN {X 0,Y 566.223,Z 334.572,A -85,B 0,C 180,E1 -2559.273,E2 -2559.273} C_VEL
LIN {X 0,Y 566.211,Z 334.573,A -85,B 0,C 180,E1 -2562.087,E2 -2562.087} C_VEL
LIN {X 0,Y 566.174,Z 334.586,A -85,B 0,C 180,E1 -2565.036,E2 -2565.036} C_VEL
LIN {X 0,Y 566.213,Z 334.573,A -85,B 0,C 180,E1 -2568.136,E2 -2568.136} C_VEL
LIN {X 0,Y 566.223,Z 334.58,A -85,B 0,C 180,E1 -2570.727,E2 -2570.727} C_VEL
LIN {X 0,Y 566.184,Z 334.579,A -85,B 0,C 180,E1 -2573.788,E2 -2573.788} C_VEL
LIN {X 0,Y 566.212,Z 334.578,A -85,B 0,C 180,E1 -2576.266,E2 -2576.266} C_VEL
LIN {X 0,Y 566.199,Z 334.585,A -85,B 0,C 180,E1 -2578.922,E2 -2578.922} C_VEL
LIN {X 0,Y 566.212,Z 334.575,A -85,B 0,C 180,E1 -2581.857,E2 -2581.857} C_VEL
LIN {X 0,Y 566.23,Z 334.715,A -85,B 0,C 180,E1 -2583.274,E2 -2583.274} C_VEL
LIN {X 0,Y 567.976,Z 341.532,A -85,B 0,C 180,E1 -2584.14,E2 -2584.14} C_VEL
LIN {X 0,Y 568.139,Z 346.586,A -85,B 0,C 180,E1 -2584.696,E2 -2584.696} C_VEL
LIN {X 0,Y 567.67,Z 372.213,A -85,B 0,C 180,E1 -2587.431,E2 -2587.431} C_VEL
LIN {X 0,Y 567.291,Z 397.817,A -85,B 0,C 180,E1 -2590.107,E2 -2590.107} C_VEL
LIN {X 0,Y 568.524,Z 405.834,A -85,B 0,C 180,E1 -2590.284,E2 -2590.284} C_VEL
LIN {X 0,Y 567.977,Z 565.081,A -85,B 0,C 180,E1 -2592.366,E2 -2592.366} C_VEL
LIN {X 0,Y 567.829,Z 580.707,A -85,B 0,C 180,E1 -2592.72,E2 -2592.72} C_VEL
LIN {X 0,Y 567.615,Z 596.041,A -85,B 0,C 180,E1 -2593.223,E2 -2593.223} C_VEL
LIN {X 0,Y 567.46,Z 609.774,A -85,B 0,C 180,E1 -2593.82,E2 -2593.82} C_VEL
LIN {X 0,Y 567.146,Z 623.247,A -85,B 0,C 180,E1 -2594.548,E2 -2594.548} C_VEL
LIN {X 0,Y 566.922,Z 636.502,A -85,B 0,C 180,E1 -2595.429,E2 -2595.429} C_VEL
LIN {X 0,Y 566.674,Z 649.351,A -85,B 0,C 180,E1 -2596.462,E2 -2596.462} C_VEL
LIN {X 0,Y 566.491,Z 659.75,A -85,B 0,C 180,E1 -2597.461,E2 -2597.461} C_VEL
LIN {X 0,Y 566.268,Z 670.313,A -85,B 0,C 180,E1 -2598.659,E2 -2598.659} C_VEL
LIN {X 0,Y 566.209,Z 678.857,A -85,B 0,C 180,E1 -2599.812,E2 -2599.812} C_VEL
LIN {X 0,Y 566.056,Z 686.734,A -85,B 0,C 180,E1 -2601.072,E2 -2601.072} C_VEL
LIN {X 0,Y 565.997,Z 694.09,A -85,B 0,C 180,E1 -2602.509,E2 -2602.509} C_VEL
LIN {X 0,Y 565.958,Z 699.923,A -85,B 0,C 180,E1 -2603.941,E2 -2603.941} C_VEL
LIN {X 0,Y 565.866,Z 703.386,A -85,B 0,C 180,E1 -2605.013,E2 -2605.013} C_VEL
LIN {X 0,Y 565.91,Z 706.89,A -85,B 0,C 180,E1 -2606.44,E2 -2606.44} C_VEL
LIN {X 0,Y 565.839,Z 709.192,A -85,B 0,C 180,E1 -2607.865,E2 -2607.865} C_VEL
LIN {X 0,Y 565.836,Z 710.349,A -85,B 0,C 180,E1 -2609.288,E2 -2609.288} C_VEL
LIN {X 0,Y 565.837,Z 710.349,A -85,B 0,C 180,E1 -2610.712,E2 -2610.712} C_VEL
LIN {X 0,Y 565.838,Z 709.19,A -85,B 0,C 180,E1 -2612.136,E2 -2612.136} C_VEL
LIN {X 0,Y 565.91,Z 706.887,A -85,B 0,C 180,E1 -2613.56,E2 -2613.56} C_VEL
LIN {X 0,Y 565.866,Z 703.385,A -85,B 0,C 180,E1 -2614.988,E2 -2614.988} C_VEL
LIN {X 0,Y 565.943,Z 698.608,A -85,B 0,C 180,E1 -2616.417,E2 -2616.417} C_VEL
LIN {X 0,Y 566.015,Z 692.422,A -85,B 0,C 180,E1 -2617.85,E2 -2617.85} C_VEL
LIN {X 0,Y 566.071,Z 684.647,A -85,B 0,C 180,E1 -2619.288,E2 -2619.288} C_VEL
LIN {X 0,Y 566.239,Z 676.368,A -85,B 0,C 180,E1 -2620.549,E2 -2620.549} C_VEL
LIN {X 0,Y 566.367,Z 666.39,A -85,B 0,C 180,E1 -2621.815,E2 -2621.815} C_VEL
LIN {X 0,Y 566.586,Z 656.187,A -85,B 0,C 180,E1 -2622.902,E2 -2622.902} C_VEL
LIN {X 0,Y 566.763,Z 644.018,A -85,B 0,C 180,E1 -2623.993,E2 -2623.993} C_VEL
LIN {X 0,Y 567.039,Z 631.338,A -85,B 0,C 180,E1 -2624.936,E2 -2624.936} C_VEL
LIN {X 0,Y 567.229,Z 618.511,A -85,B 0,C 180,E1 -2625.726,E2 -2625.726} C_VEL
LIN {X 0,Y 567.504,Z 603.826,A -85,B 0,C 180,E1 -2626.457,E2 -2626.457} C_VEL
LIN {X 0,Y 567.707,Z 589.611,A -85,B 0,C 180,E1 -2627.006,E2 -2627.006} C_VEL
LIN {X 0,Y 567.904,Z 574.285,A -85,B 0,C 180,E1 -2627.442,E2 -2627.442} C_VEL
LIN {X 0,Y 567.998,Z 559.614,A -85,B 0,C 180,E1 -2627.718,E2 -2627.718} C_VEL
LIN {X 0,Y 568.414,Z 404.152,A -85,B 0,C 180,E1 -2629.742,E2 -2629.742} C_VEL
LIN {X 0,Y 567.281,Z 397.897,A -85,B 0,C 180,E1 -2629.888,E2 -2629.888} C_VEL
LIN {X 0,Y 567.671,Z 372.211,A -85,B 0,C 180,E1 -2632.569,E2 -2632.569} C_VEL
LIN {X 0,Y 568.171,Z 345.165,A -85,B 0,C 180,E1 -2635.448,E2 -2635.448} C_VEL
LIN {X 0,Y 567.958,Z 341.454,A -85,B 0,C 180,E1 -2635.861,E2 -2635.861} C_VEL
LIN {X 0,Y 566.23,Z 334.681,A -85,B 0,C 180,E1 -2636.725,E2 -2636.725} C_VEL
LIN {X 0,Y 566.204,Z 334.581,A -85,B 0,C 180,E1 -2639.672,E2 -2639.672} C_VEL
LIN {X 0,Y 566.204,Z 334.58,A -85,B 0,C 180,E1 -2642.43,E2 -2642.43} C_VEL
LIN {X 0,Y 566.202,Z 334.586,A -85,B 0,C 180,E1 -2644.993,E2 -2644.993} C_VEL
LIN {X 0,Y 566.198,Z 334.58,A -85,B 0,C 180,E1 -2647.461,E2 -2647.461} C_VEL
LIN {X 0,Y 566.208,Z 334.579,A -85,B 0,C 180,E1 -2650.199,E2 -2650.199} C_VEL
LIN {X 0,Y 566.198,Z 334.582,A -85,B 0,C 180,E1 -2653.055,E2 -2653.055} C_VEL
LIN {X 0,Y 566.194,Z 334.58,A -85,B 0,C 180,E1 -2656.049,E2 -2656.049} C_VEL
LIN {X 0,Y 566.204,Z 334.578,A -85,B 0,C 180,E1 -2659.215,E2 -2659.215} C_VEL
LIN {X 0,Y 566.181,Z 334.581,A -85,B 0,C 180,E1 -2661.636,E2 -2661.636} C_VEL
LIN {X 0,Y 566.143,Z 334.593,A -85,B 0,C 180,E1 -2664.307,E2 -2664.307} C_VEL
LIN {X 0,Y 566.208,Z 334.579,A -85,B 0,C 180,E1 -2666.897,E2 -2666.897} C_VEL
LIN {X 0,Y 566.167,Z 334.583,A -85,B 0,C 180,E1 -2669.407,E2 -2669.407} C_VEL
LIN {X 0,Y 566.14,Z 334.592,A -85,B 0,C 180,E1 -2671.854,E2 -2671.854} C_VEL
LIN {X 0,Y 566.196,Z 334.699,A -85,B 0,C 180,E1 -2674.726,E2 -2674.726} C_VEL
LIN {X 0,Y 567.53,Z 341.065,A -85,B 0,C 180,E1 -2675.685,E2 -2675.685} C_VEL
LIN {X 0,Y 567.279,Z 356.813,A -85,B 0,C 180,E1 -2677.799,E2 -2677.799} C_VEL
LIN {X 0,Y 566.981,Z 375.766,A -85,B 0,C 180,E1 -2680.278,E2 -2680.278} C_VEL
LIN {X 0,Y 566.713,Z 397.139,A -85,B 0,C 180,E1 -2683.019,E2 -2683.019} C_VEL
LIN {X 0,Y 567.015,Z 399.305,A -85,B 0,C 180,E1 -2683.104,E2 -2683.104} C_VEL
LIN {X 0,Y 567.797,Z 404.504,A -85,B 0,C 180,E1 -2683.195,E2 -2683.195} C_VEL
LIN {X 0,Y 567.424,Z 535.993,A -85,B 0,C 180,E1 -2684.901,E2 -2684.901} C_VEL
LIN {X 0,Y 567.32,Z 550.368,A -85,B 0,C 180,E1 -2685.24,E2 -2685.24} C_VEL
LIN {X 0,Y 567.134,Z 564.87,A -85,B 0,C 180,E1 -2685.742,E2 -2685.742} C_VEL
LIN {X 0,Y 566.947,Z 578.499,A -85,B 0,C 180,E1 -2686.377,E2 -2686.377} C_VEL
LIN {X 0,Y 566.744,Z 590.808,A -85,B 0,C 180,E1 -2687.102,E2 -2687.102} C_VEL
LIN {X 0,Y 566.578,Z 602.033,A -85,B 0,C 180,E1 -2687.917,E2 -2687.917} C_VEL
LIN {X 0,Y 566.452,Z 612.791,A -85,B 0,C 180,E1 -2688.856,E2 -2688.856} C_VEL
LIN {X 0,Y 566.248,Z 621.895,A -85,B 0,C 180,E1 -2689.813,E2 -2689.813} C_VEL
LIN {X 0,Y 566.151,Z 630.582,A -85,B 0,C 180,E1 -2690.893,E2 -2690.893} C_VEL
LIN {X 0,Y 566.06,Z 638.819,A -85,B 0,C 180,E1 -2692.151,E2 -2692.151} C_VEL
LIN {X 0,Y 565.967,Z 645.606,A -85,B 0,C 180,E1 -2693.422,E2 -2693.422} C_VEL
LIN {X 0,Y 565.928,Z 650.768,A -85,B 0,C 180,E1 -2694.656,E2 -2694.656} C_VEL
LIN {X 0,Y 565.957,Z 654.294,A -85,B 0,C 180,E1 -2695.727,E2 -2695.727} C_VEL
LIN {X 0,Y 565.875,Z 657.755,A -85,B 0,C 180,E1 -2697.153,E2 -2697.153} C_VEL
LIN {X 0,Y 565.844,Z 659.763,A -85,B 0,C 180,E1 -2698.577,E2 -2698.577} C_VEL
LIN {X 0,Y 565.838,Z 660.496,A -85,B 0,C 180,E1 -2700,E2 -2700} C_VEL
LIN {X 0,Y 565.841,Z 659.846,A -85,B 0,C 180,E1 -2701.424,E2 -2701.424} C_VEL
LIN {X 0,Y 565.873,Z 657.929,A -85,B 0,C 180,E1 -2702.848,E2 -2702.848} C_VEL
LIN {X 0,Y 565.957,Z 654.559,A -85,B 0,C 180,E1 -2704.273,E2 -2704.273} C_VEL
LIN {X 0,Y 565.985,Z 649.764,A -85,B 0,C 180,E1 -2705.701,E2 -2705.701} C_VEL
LIN {X 0,Y 565.996,Z 645.246,A -85,B 0,C 180,E1 -2706.739,E2 -2706.739} C_VEL
LIN {X 0,Y 566.044,Z 638.304,A -85,B 0,C 180,E1 -2708.029,E2 -2708.029} C_VEL
LIN {X 0,Y 566.172,Z 629.878,A -85,B 0,C 180,E1 -2709.287,E2 -2709.287} C_VEL
LIN {X 0,Y 566.294,Z 621.129,A -85,B 0,C 180,E1 -2710.367,E2 -2710.367} C_VEL
LIN {X 0,Y 566.487,Z 610.463,A -85,B 0,C 180,E1 -2711.449,E2 -2711.449} C_VEL
LIN {X 0,Y 566.619,Z 599.73,A -85,B 0,C 180,E1 -2712.355,E2 -2712.355} C_VEL
LIN {X 0,Y 566.797,Z 587.953,A -85,B 0,C 180,E1 -2713.17,E2 -2713.17} C_VEL
LIN {X 0,Y 567.02,Z 574.993,A -85,B 0,C 180,E1 -2713.895,E2 -2713.895} C_VEL
LIN {X 0,Y 567.204,Z 562.151,A -85,B 0,C 180,E1 -2714.455,E2 -2714.455} C_VEL
LIN {X 0,Y 567.328,Z 548.21,A -85,B 0,C 180,E1 -2714.909,E2 -2714.909} C_VEL
LIN {X 0,Y 567.432,Z 534.434,A -85,B 0,C 180,E1 -2715.214,E2 -2715.214} C_VEL
LIN {X 0,Y 567.626,Z 473.907,A -85,B 0,C 180,E1 -2716.003,E2 -2716.003} C_VEL
LIN {X 0,Y 566.99,Z 468.102,A -85,B 0,C 180,E1 -2716.097,E2 -2716.097} C_VEL
LIN {X 0,Y 561.481,Z 449.456,A -85,B 0,C 180,E1 -2716.502,E2 -2716.502} C_VEL
LIN {X 0,Y 560.898,Z 443.651,A -85,B 0,C 180,E1 -2716.595,E2 -2716.595} C_VEL
LIN {X 0,Y 560.891,Z 403.875,A -85,B 0,C 180,E1 -2717.117,E2 -2717.117} C_VEL
LIN {X 0,Y 559.74,Z 397.357,A -85,B 0,C 180,E1 -2717.266,E2 -2717.266} C_VEL
LIN {X 0,Y 560.091,Z 376.305,A -85,B 0,C 180,E1 -2719.995,E2 -2719.995} C_VEL
LIN {X 0,Y 560.578,Z 351.764,A -85,B 0,C 180,E1 -2723.261,E2 -2723.261} C_VEL
LIN {X 0,Y 560.69,Z 343.095,A -85,B 0,C 180,E1 -2724.434,E2 -2724.434} C_VEL
LIN {X 0,Y 559.158,Z 335.568,A -85,B 0,C 180,E1 -2725.573,E2 -2725.573} C_VEL
LIN {X 0,Y 559.097,Z 335.466,A -85,B 0,C 180,E1 -2728.533,E2 -2728.533} C_VEL
LIN {X 0,Y 559.118,Z 335.46,A -85,B 0,C 180,E1 -2731.268,E2 -2731.268} C_VEL
LIN {X 0,Y 559.14,Z 335.465,A -85,B 0,C 180,E1 -2733.945,E2 -2733.945} C_VEL
LIN {X 0,Y 559.103,Z 335.461,A -85,B 0,C 180,E1 -2737.111,E2 -2737.111} C_VEL
LIN {X 0,Y 559.119,Z 335.467,A -85,B 0,C 180,E1 -2739.936,E2 -2739.936} C_VEL
LIN {X 0,Y 559.109,Z 335.458,A -85,B 0,C 180,E1 -2742.749,E2 -2742.749} C_VEL
LIN {X 0,Y 559.112,Z 335.465,A -85,B 0,C 180,E1 -2745.765,E2 -2745.765} C_VEL
LIN {X 0,Y 559.092,Z 335.47,A -85,B 0,C 180,E1 -2748.223,E2 -2748.223} C_VEL
LIN {X 0,Y 559.135,Z 335.456,A -85,B 0,C 180,E1 -2751.197,E2 -2751.197} C_VEL
LIN {X 0,Y 559.106,Z 335.465,A -85,B 0,C 180,E1 -2753.787,E2 -2753.787} C_VEL
LIN {X 0,Y 559.123,Z 335.464,A -85,B 0,C 180,E1 -2756.422,E2 -2756.422} C_VEL
LIN {X 0,Y 559.139,Z 335.458,A -85,B 0,C 180,E1 -2758.979,E2 -2758.979} C_VEL
LIN {X 0,Y 559.158,Z 335.568,A -85,B 0,C 180,E1 -2762.386,E2 -2762.386} C_VEL
LIN {X 0,Y 561.184,Z 344.751,A -85,B 0,C 180,E1 -2763.603,E2 -2763.603} C_VEL
LIN {X 0,Y 560.826,Z 366.657,A -85,B 0,C 180,E1 -2766.178,E2 -2766.178} C_VEL
LIN {X 0,Y 560.436,Z 391.156,A -85,B 0,C 180,E1 -2769.059,E2 -2769.059} C_VEL
LIN {X 0,Y 560.268,Z 398.548,A -85,B 0,C 180,E1 -2769.907,E2 -2769.907} C_VEL
LIN {X 0,Y 561.823,Z 407.217,A -85,B 0,C 180,E1 -2770.103,E2 -2770.103} C_VEL
LIN {X 0,Y 561.2,Z 563.792,A -85,B 0,C 180,E1 -2772.176,E2 -2772.176} C_VEL
LIN {X 0,Y 561.071,Z 577.86,A -85,B 0,C 180,E1 -2772.477,E2 -2772.477} C_VEL
LIN {X 0,Y 560.842,Z 593.622,A -85,B 0,C 180,E1 -2772.967,E2 -2772.967} C_VEL
LIN {X 0,Y 560.632,Z 606.812,A -85,B 0,C 180,E1 -2773.523,E2 -2773.523} C_VEL
LIN {X 0,Y 560.365,Z 619.252,A -85,B 0,C 180,E1 -2774.17,E2 -2774.17} C_VEL
LIN {X 0,Y 560.118,Z 630.916,A -85,B 0,C 180,E1 -2774.898,E2 -2774.898} C_VEL
LIN {X 0,Y 559.841,Z 642.269,A -85,B 0,C 180,E1 -2775.737,E2 -2775.737} C_VEL
LIN {X 0,Y 559.599,Z 653.834,A -85,B 0,C 180,E1 -2776.75,E2 -2776.75} C_VEL
LIN {X 0,Y 559.389,Z 664.382,A -85,B 0,C 180,E1 -2777.852,E2 -2777.852} C_VEL
LIN {X 0,Y 559.226,Z 673.225,A -85,B 0,C 180,E1 -2778.941,E2 -2778.941} C_VEL
LIN {X 0,Y 559.094,Z 680.944,A -85,B 0,C 180,E1 -2780.047,E2 -2780.047} C_VEL
LIN {X 0,Y 559.002,Z 688.462,A -85,B 0,C 180,E1 -2781.323,E2 -2781.323} C_VEL
LIN {X 0,Y 558.901,Z 695.514,A -85,B 0,C 180,E1 -2782.776,E2 -2782.776} C_VEL
LIN {X 0,Y 558.887,Z 701.025,A -85,B 0,C 180,E1 -2784.226,E2 -2784.226} C_VEL
LIN {X 0,Y 558.809,Z 705.159,A -85,B 0,C 180,E1 -2785.672,E2 -2785.672} C_VEL
LIN {X 0,Y 558.793,Z 708.102,A -85,B 0,C 180,E1 -2787.116,E2 -2787.116} C_VEL
LIN {X 0,Y 558.742,Z 709.874,A -85,B 0,C 180,E1 -2788.558,E2 -2788.558} C_VEL
LIN {X 0,Y 558.738,Z 710.496,A -85,B 0,C 180,E1 -2790,E2 -2790} C_VEL
LIN {X 0,Y 558.743,Z 709.96,A -85,B 0,C 180,E1 -2791.441,E2 -2791.441} C_VEL
LIN {X 0,Y 558.795,Z 708.255,A -85,B 0,C 180,E1 -2792.884,E2 -2792.884} C_VEL
LIN {X 0,Y 558.809,Z 705.375,A -85,B 0,C 180,E1 -2794.328,E2 -2794.328} C_VEL
LIN {X 0,Y 558.887,Z 701.307,A -85,B 0,C 180,E1 -2795.774,E2 -2795.774} C_VEL
LIN {X 0,Y 558.899,Z 695.912,A -85,B 0,C 180,E1 -2797.224,E2 -2797.224} C_VEL
LIN {X 0,Y 558.988,Z 688.958,A -85,B 0,C 180,E1 -2798.677,E2 -2798.677} C_VEL
LIN {X 0,Y 559.091,Z 681.52,A -85,B 0,C 180,E1 -2799.953,E2 -2799.953} C_VEL
LIN {X 0,Y 559.2,Z 673.89,A -85,B 0,C 180,E1 -2801.059,E2 -2801.059} C_VEL
LIN {X 0,Y 559.381,Z 665.144,A -85,B 0,C 180,E1 -2802.148,E2 -2802.148} C_VEL
LIN {X 0,Y 559.619,Z 654.776,A -85,B 0,C 180,E1 -2803.25,E2 -2803.25} C_VEL
LIN {X 0,Y 559.846,Z 642.236,A -85,B 0,C 180,E1 -2804.355,E2 -2804.355} C_VEL
LIN {X 0,Y 560.127,Z 631.556,A -85,B 0,C 180,E1 -2805.148,E2 -2805.148} C_VEL
LIN {X 0,Y 560.302,Z 620.8,A -85,B 0,C 180,E1 -2805.832,E2 -2805.832} C_VEL
LIN {X 0,Y 560.59,Z 608.645,A -85,B 0,C 180,E1 -2806.478,E2 -2806.478} C_VEL
LIN {X 0,Y 560.786,Z 597.003,A -85,B 0,C 180,E1 -2806.987,E2 -2806.987} C_VEL
LIN {X 0,Y 561.027,Z 582.963,A -85,B 0,C 180,E1 -2807.473,E2 -2807.473} C_VEL
LIN {X 0,Y 561.184,Z 566.803,A -85,B 0,C 180,E1 -2807.864,E2 -2807.864} C_VEL
LIN {X 0,Y 561.332,Z 538.527,A -85,B 0,C 180,E1 -2808.264,E2 -2808.264} C_VEL
LIN {X 0,Y 561.827,Z 407.525,A -85,B 0,C 180,E1 -2809.983,E2 -2809.983} C_VEL
LIN {X 0,Y 560.307,Z 398.532,A -85,B 0,C 180,E1 -2810.183,E2 -2810.183} C_VEL
LIN {X 0,Y 560.762,Z 373.943,A -85,B 0,C 180,E1 -2813.057,E2 -2813.057} C_VEL
LIN {X 0,Y 561.13,Z 348.871,A -85,B 0,C 180,E1 -2816,E2 -2816} C_VEL
LIN {X 0,Y 561.095,Z 343.806,A -85,B 0,C 180,E1 -2816.602,E2 -2816.602} C_VEL
LIN {X 0,Y 559.161,Z 335.61,A -85,B 0,C 180,E1 -2817.687,E2 -2817.687} C_VEL
LIN {X 0,Y 559.138,Z 335.458,A -85,B 0,C 180,E1 -2821.02,E2 -2821.02} C_VEL
LIN {X 0,Y 559.139,Z 335.463,A -85,B 0,C 180,E1 -2823.945,E2 -2823.945} C_VEL
LIN {X 0,Y 559.104,Z 335.461,A -85,B 0,C 180,E1 -2827.111,E2 -2827.111} C_VEL
LIN {X 0,Y 559.119,Z 335.464,A -85,B 0,C 180,E1 -2829.936,E2 -2829.936} C_VEL
LIN {X 0,Y 559.11,Z 335.459,A -85,B 0,C 180,E1 -2832.748,E2 -2832.748} C_VEL
LIN {X 0,Y 559.123,Z 335.466,A -85,B 0,C 180,E1 -2835.764,E2 -2835.764} C_VEL
LIN {X 0,Y 559.098,Z 335.465,A -85,B 0,C 180,E1 -2838.224,E2 -2838.224} C_VEL
LIN {X 0,Y 559.167,Z 335.453,A -85,B 0,C 180,E1 -2841.193,E2 -2841.193} C_VEL
LIN {X 0,Y 559.114,Z 335.467,A -85,B 0,C 180,E1 -2843.787,E2 -2843.787} C_VEL
LIN {X 0,Y 559.146,Z 335.456,A -85,B 0,C 180,E1 -2846.424,E2 -2846.424} C_VEL
LIN {X 0,Y 559.151,Z 335.453,A -85,B 0,C 180,E1 -2848.98,E2 -2848.98} C_VEL
LIN {X 0,Y 559.134,Z 335.466,A -85,B 0,C 180,E1 -2851.626,E2 -2851.626} C_VEL
LIN {X 0,Y 559.139,Z 335.456,A -85,B 0,C 180,E1 -2854.822,E2 -2854.822} C_VEL
LIN {X 0,Y 559.139,Z 335.46,A -85,B 0,C 180,E1 -2857.847,E2 -2857.847} C_VEL
LIN {X 0,Y 559.193,Z 335.449,A -85,B 0,C 180,E1 -2860.494,E2 -2860.494} C_VEL
LIN {X 0,Y 559.168,Z 335.454,A -85,B 0,C 180,E1 -2863.197,E2 -2863.197} C_VEL
LIN {X 0,Y 559.167,Z 335.454,A -85,B 0,C 180,E1 -2866.184,E2 -2866.184} C_VEL
LIN {X 0,Y 559.193,Z 335.45,A -85,B 0,C 180,E1 -2869.133,E2 -2869.133} C_VEL
LIN {X 0,Y 559.181,Z 335.453,A -85,B 0,C 180,E1 -2872.053,E2 -2872.053} C_VEL
LIN {X 0,Y 559.248,Z 335.442,A -85,B 0,C 180,E1 -2874.953,E2 -2874.953} C_VEL
LIN {X 0,Y 559.255,Z 335.445,A -85,B 0,C 180,E1 -2877.839,E2 -2877.839} C_VEL
LIN {X 0,Y 559.264,Z 335.439,A -85,B 0,C 180,E1 -2880.72,E2 -2880.72} C_VEL
LIN {X 0,Y 559.23,Z 335.444,A -85,B 0,C 180,E1 -2882.881,E2 -2882.881} C_VEL
LIN {X 0,Y 559.23,Z 335.447,A -85,B 0,C 180,E1 -2885.77,E2 -2885.77} C_VEL
LIN {X 0,Y 559.17,Z 335.45,A -85,B 0,C 180,E1 -2888.675,E2 -2888.675} C_VEL
LIN {X 0,Y 559.207,Z 335.451,A -85,B 0,C 180,E1 -2891.6,E2 -2891.6} C_VEL
LIN {X 0,Y 559.181,Z 335.448,A -85,B 0,C 180,E1 -2894.587,E2 -2894.587} C_VEL
LIN {X 0,Y 559.143,Z 335.459,A -85,B 0,C 180,E1 -2897.557,E2 -2897.557} C_VEL
LIN {X 0,Y 559.166,Z 335.452,A -85,B 0,C 180,E1 -2899.838,E2 -2899.838} C_VEL
LIN {X 0,Y 559.141,Z 335.456,A -85,B 0,C 180,E1 -2902.153,E2 -2902.153} C_VEL
LIN {X 0,Y 559.177,Z 335.458,A -85,B 0,C 180,E1 -2905.298,E2 -2905.298} C_VEL
LIN {X 0,Y 559.157,Z 335.456,A -85,B 0,C 180,E1 -2907.713,E2 -2907.713} C_VEL
LIN {X 0,Y 559.155,Z 335.451,A -85,B 0,C 180,E1 -2910.183,E2 -2910.183} C_VEL
LIN {X 0,Y 559.157,Z 335.458,A -85,B 0,C 180,E1 -2912.715,E2 -2912.715} C_VEL
LIN {X 0,Y 559.128,Z 335.463,A -85,B 0,C 180,E1 -2915.324,E2 -2915.324} C_VEL
LIN {X 0,Y 559.136,Z 335.455,A -85,B 0,C 180,E1 -2918.017,E2 -2918.017} C_VEL
LIN {X 0,Y 559.176,Z 335.449,A -85,B 0,C 180,E1 -2920.811,E2 -2920.811} C_VEL
LIN {X 0,Y 559.142,Z 335.457,A -85,B 0,C 180,E1 -2923.734,E2 -2923.734} C_VEL
LIN {X 0,Y 559.146,Z 335.457,A -85,B 0,C 180,E1 -2926.803,E2 -2926.803} C_VEL
LIN {X 0,Y 559.176,Z 335.458,A -85,B 0,C 180,E1 -2929.189,E2 -2929.189} C_VEL
LIN {X 0,Y 559.135,Z 335.457,A -85,B 0,C 180,E1 -2931.983,E2 -2931.983} C_VEL
LIN {X 0,Y 559.132,Z 335.466,A -85,B 0,C 180,E1 -2934.787,E2 -2934.787} C_VEL
LIN {X 0,Y 559.157,Z 335.457,A -85,B 0,C 180,E1 -2937.364,E2 -2937.364} C_VEL
LIN {X 0,Y 559.15,Z 335.459,A -85,B 0,C 180,E1 -2940.142,E2 -2940.142} C_VEL
LIN {X 0,Y 559.17,Z 335.569,A -85,B 0,C 180,E1 -2942.997,E2 -2942.997} C_VEL
LIN {X 0,Y 559.948,Z 338.516,A -85,B 0,C 180,E1 -2943.413,E2 -2943.413} C_VEL
LIN {X 0,Y 561.363,Z 344.298,A -85,B 0,C 180,E1 -2944.128,E2 -2944.128} C_VEL
LIN {X 0,Y 561.016,Z 364.964,A -85,B 0,C 180,E1 -2946.367,E2 -2946.367} C_VEL
LIN {X 0,Y 560.526,Z 392.008,A -85,B 0,C 180,E1 -2949.255,E2 -2949.255} C_VEL
LIN {X 0,Y 560.483,Z 398.034,A -85,B 0,C 180,E1 -2949.867,E2 -2949.867} C_VEL
LIN {X 0,Y 561.84,Z 406.223,A -85,B 0,C 180,E1 -2950.045,E2 -2950.045} C_VEL
LIN {X 0,Y 561.222,Z 565.2,A -85,B 0,C 180,E1 -2952.149,E2 -2952.149} C_VEL
LIN {X 0,Y 561.066,Z 580.705,A -85,B 0,C 180,E1 -2952.505,E2 -2952.505} C_VEL
LIN {X 0,Y 560.799,Z 596.039,A -85,B 0,C 180,E1 -2953.013,E2 -2953.013} C_VEL
LIN {X 0,Y 560.617,Z 609.777,A -85,B 0,C 180,E1 -2953.617,E2 -2953.617} C_VEL
LIN {X 0,Y 560.259,Z 623.249,A -85,B 0,C 180,E1 -2954.354,E2 -2954.354} C_VEL
LIN {X 0,Y 560.001,Z 636.286,A -85,B 0,C 180,E1 -2955.229,E2 -2955.229} C_VEL
LIN {X 0,Y 559.722,Z 648.293,A -85,B 0,C 180,E1 -2956.198,E2 -2956.198} C_VEL
LIN {X 0,Y 559.516,Z 659.75,A -85,B 0,C 180,E1 -2957.302,E2 -2957.302} C_VEL
LIN {X 0,Y 559.304,Z 669.39,A -85,B 0,C 180,E1 -2958.402,E2 -2958.402} C_VEL
LIN {X 0,Y 559.168,Z 678.857,A -85,B 0,C 180,E1 -2959.683,E2 -2959.683} C_VEL
LIN {X 0,Y 559.002,Z 686.735,A -85,B 0,C 180,E1 -2960.958,E2 -2960.958} C_VEL
LIN {X 0,Y 558.92,Z 694.09,A -85,B 0,C 180,E1 -2962.413,E2 -2962.413} C_VEL
LIN {X 0,Y 558.859,Z 699.923,A -85,B 0,C 180,E1 -2963.864,E2 -2963.864} C_VEL
LIN {X 0,Y 558.787,Z 703.386,A -85,B 0,C 180,E1 -2964.949,E2 -2964.949} C_VEL
LIN {X 0,Y 558.819,Z 706.889,A -85,B 0,C 180,E1 -2966.395,E2 -2966.395} C_VEL
LIN {X 0,Y 558.744,Z 709.191,A -85,B 0,C 180,E1 -2967.838,E2 -2967.838} C_VEL
LIN {X 0,Y 558.737,Z 710.349,A -85,B 0,C 180,E1 -2969.279,E2 -2969.279} C_VEL
LIN {X 0,Y 558.737,Z 710.348,A -85,B 0,C 180,E1 -2970.721,E2 -2970.721} C_VEL
LIN {X 0,Y 558.744,Z 709.189,A -85,B 0,C 180,E1 -2972.163,E2 -2972.163} C_VEL
LIN {X 0,Y 558.819,Z 706.886,A -85,B 0,C 180,E1 -2973.605,E2 -2973.605} C_VEL
LIN {X 0,Y 558.787,Z 703.386,A -85,B 0,C 180,E1 -2975.051,E2 -2975.051} C_VEL
LIN {X 0,Y 558.85,Z 698.608,A -85,B 0,C 180,E1 -2976.499,E2 -2976.499} C_VEL
LIN {X 0,Y 558.951,Z 692.421,A -85,B 0,C 180,E1 -2977.95,E2 -2977.95} C_VEL
LIN {X 0,Y 559.005,Z 684.646,A -85,B 0,C 180,E1 -2979.407,E2 -2979.407} C_VEL
LIN {X 0,Y 559.217,Z 676.367,A -85,B 0,C 180,E1 -2980.683,E2 -2980.683} C_VEL
LIN {X 0,Y 559.363,Z 666.39,A -85,B 0,C 180,E1 -2981.965,E2 -2981.965} C_VEL
LIN {X 0,Y 559.596,Z 656.186,A -85,B 0,C 180,E1 -2983.066,E2 -2983.066} C_VEL
LIN {X 0,Y 559.825,Z 644.018,A -85,B 0,C 180,E1 -2984.17,E2 -2984.17} C_VEL
LIN {X 0,Y 560.123,Z 631.686,A -85,B 0,C 180,E1 -2985.1,E2 -2985.1} C_VEL
LIN {X 0,Y 560.358,Z 618.508,A -85,B 0,C 180,E1 -2985.924,E2 -2985.924} C_VEL
LIN {X 0,Y 560.666,Z 603.824,A -85,B 0,C 180,E1 -2986.663,E2 -2986.663} C_VEL
LIN {X 0,Y 560.914,Z 589.61,A -85,B 0,C 180,E1 -2987.218,E2 -2987.218} C_VEL
LIN {X 0,Y 561.133,Z 574.15,A -85,B 0,C 180,E1 -2987.663,E2 -2987.663} C_VEL
LIN {X 0,Y 561.249,Z 559.264,A -85,B 0,C 180,E1 -2987.944,E2 -2987.944} C_VEL
LIN {X 0,Y 561.765,Z 405.081,A -85,B 0,C 180,E1 -2989.973,E2 -2989.973} C_VEL
LIN {X 0,Y 560.473,Z 397.827,A -85,B 0,C 180,E1 -2990.146,E2 -2990.146} C_VEL
LIN {X 0,Y 560.908,Z 370.36,A -85,B 0,C 180,E1 -2993.051,E2 -2993.051} C_VEL
LIN {X 0,Y 561.425,Z 345.218,A -85,B 0,C 180,E1 -2995.754,E2 -2995.754} C_VEL
LIN {X 0,Y 559.588,Z 337.221,A -85,B 0,C 180,E1 -2996.735,E2 -2996.735} C_VEL
LIN {X 0,Y 559.193,Z 335.566,A -85,B 0,C 180,E1 -2996.977,E2 -2996.977} C_VEL
LIN {X 0,Y 559.15,Z 335.459,A -85,B 0,C 180,E1 -2999.858,E2 -2999.858} C_VEL
LIN {X 0,Y 559.157,Z 335.462,A -85,B 0,C 180,E1 -3002.715,E2 -3002.715} C_VEL
LIN {X 0,Y 559.145,Z 335.461,A -85,B 0,C 180,E1 -3005.323,E2 -3005.323} C_VEL
LIN {X 0,Y 559.134,Z 335.459,A -85,B 0,C 180,E1 -3008.018,E2 -3008.018} C_VEL
LIN {X 0,Y 559.156,Z 335.463,A -85,B 0,C 180,E1 -3010.813,E2 -3010.813} C_VEL
LIN {X 0,Y 559.138,Z 335.458,A -85,B 0,C 180,E1 -3013.734,E2 -3013.734} C_VEL
LIN {X 0,Y 559.142,Z 335.463,A -85,B 0,C 180,E1 -3016.804,E2 -3016.804} C_VEL
LIN {X 0,Y 559.156,Z 335.457,A -85,B 0,C 180,E1 -3019.188,E2 -3019.188} C_VEL
LIN {X 0,Y 559.129,Z 335.462,A -85,B 0,C 180,E1 -3021.982,E2 -3021.982} C_VEL
LIN {X 0,Y 559.124,Z 335.463,A -85,B 0,C 180,E1 -3024.789,E2 -3024.789} C_VEL
LIN {X 0,Y 559.151,Z 335.457,A -85,B 0,C 180,E1 -3027.366,E2 -3027.366} C_VEL
LIN {X 0,Y 559.112,Z 335.469,A -85,B 0,C 180,E1 -3030.15,E2 -3030.15} C_VEL
LIN {X 0,Y 559.111,Z 335.465,A -85,B 0,C 180,E1 -3033.185,E2 -3033.185} C_VEL
LIN {X 0,Y 559.155,Z 335.688,A -85,B 0,C 180,E1 -3034.527,E2 -3034.527} C_VEL
LIN {X 0,Y 560.677,Z 342.633,A -85,B 0,C 180,E1 -3035.566,E2 -3035.566} C_VEL
LIN {X 0,Y 560.494,Z 355.549,A -85,B 0,C 180,E1 -3037.321,E2 -3037.321} C_VEL
LIN {X 0,Y 560.119,Z 374.183,A -85,B 0,C 180,E1 -3039.815,E2 -3039.815} C_VEL
LIN {X 0,Y 559.764,Z 396.466,A -85,B 0,C 180,E1 -3042.725,E2 -3042.725} C_VEL
LIN {X 0,Y 559.851,Z 398.134,A -85,B 0,C 180,E1 -3042.857,E2 -3042.857} C_VEL
LIN {X 0,Y 561.021,Z 405.783,A -85,B 0,C 180,E1 -3043.002,E2 -3043.002} C_VEL
LIN {X 0,Y 560.585,Z 536.027,A -85,B 0,C 180,E1 -3044.712,E2 -3044.712} C_VEL
LIN {X 0,Y 560.456,Z 550.911,A -85,B 0,C 180,E1 -3045.07,E2 -3045.07} C_VEL
LIN {X 0,Y 560.241,Z 564.876,A -85,B 0,C 180,E1 -3045.563,E2 -3045.563} C_VEL
LIN {X 0,Y 560.041,Z 578.505,A -85,B 0,C 180,E1 -3046.206,E2 -3046.206} C_VEL
LIN {X 0,Y 559.807,Z 590.805,A -85,B 0,C 180,E1 -3046.94,E2 -3046.94} C_VEL
LIN {X 0,Y 559.602,Z 602.036,A -85,B 0,C 180,E1 -3047.765,E2 -3047.765} C_VEL
LIN {X 0,Y 559.445,Z 613.242,A -85,B 0,C 180,E1 -3048.761,E2 -3048.761} C_VEL
LIN {X 0,Y 559.239,Z 621.893,A -85,B 0,C 180,E1 -3049.684,E2 -3049.684} C_VEL
LIN {X 0,Y 559.116,Z 630.587,A -85,B 0,C 180,E1 -3050.778,E2 -3050.778} C_VEL
LIN {X 0,Y 558.982,Z 638.816,A -85,B 0,C 180,E1 -3052.051,E2 -3052.051} C_VEL
LIN {X 0,Y 558.873,Z 646.338,A -85,B 0,C 180,E1 -3053.502,E2 -3053.502} C_VEL
LIN {X 0,Y 558.858,Z 650.765,A -85,B 0,C 180,E1 -3054.588,E2 -3054.588} C_VEL
LIN {X 0,Y 558.866,Z 654.292,A -85,B 0,C 180,E1 -3055.673,E2 -3055.673} C_VEL
LIN {X 0,Y 558.796,Z 657.759,A -85,B 0,C 180,E1 -3057.116,E2 -3057.116} C_VEL
LIN {X 0,Y 558.743,Z 659.758,A -85,B 0,C 180,E1 -3058.559,E2 -3058.559} C_VEL
LIN {X 0,Y 558.739,Z 660.496,A -85,B 0,C 180,E1 -3060,E2 -3060} C_VEL
LIN {X 0,Y 558.741,Z 659.84,A -85,B 0,C 180,E1 -3061.442,E2 -3061.442} C_VEL
LIN {X 0,Y 558.794,Z 657.928,A -85,B 0,C 180,E1 -3062.884,E2 -3062.884} C_VEL
LIN {X 0,Y 558.866,Z 654.553,A -85,B 0,C 180,E1 -3064.327,E2 -3064.327} C_VEL
LIN {X 0,Y 558.915,Z 649.765,A -85,B 0,C 180,E1 -3065.774,E2 -3065.774} C_VEL
LIN {X 0,Y 558.904,Z 645.062,A -85,B 0,C 180,E1 -3066.861,E2 -3066.861} C_VEL
LIN {X 0,Y 558.985,Z 638.295,A -85,B 0,C 180,E1 -3068.131,E2 -3068.131} C_VEL
LIN {X 0,Y 559.107,Z 629.871,A -85,B 0,C 180,E1 -3069.405,E2 -3069.405} C_VEL
LIN {X 0,Y 559.266,Z 621.117,A -85,B 0,C 180,E1 -3070.499,E2 -3070.499} C_VEL
LIN {X 0,Y 559.487,Z 610.449,A -85,B 0,C 180,E1 -3071.595,E2 -3071.595} C_VEL
LIN {X 0,Y 559.639,Z 599.724,A -85,B 0,C 180,E1 -3072.511,E2 -3072.511} C_VEL
LIN {X 0,Y 559.829,Z 587.935,A -85,B 0,C 180,E1 -3073.337,E2 -3073.337} C_VEL
LIN {X 0,Y 560.104,Z 574.974,A -85,B 0,C 180,E1 -3074.07,E2 -3074.07} C_VEL
LIN {X 0,Y 560.326,Z 562.396,A -85,B 0,C 180,E1 -3074.625,E2 -3074.625} C_VEL
LIN {X 0,Y 560.467,Z 548.599,A -85,B 0,C 180,E1 -3075.084,E2 -3075.084} C_VEL
LIN {X 0,Y 560.582,Z 534.378,A -85,B 0,C 180,E1 -3075.404,E2 -3075.404} C_VEL
LIN {X 0,Y 560.898,Z 443.651,A -85,B 0,C 180,E1 -3076.595,E2 -3076.595} C_VEL
LIN {X 0,Y 560.286,Z 437.84,A -85,B 0,C 180,E1 -3076.69,E2 -3076.69} C_VEL
LIN {X 0,Y 554.701,Z 419.212,A -85,B 0,C 180,E1 -3077.11,E2 -3077.11} C_VEL
LIN {X 0,Y 554.188,Z 413.402,A -85,B 0,C 180,E1 -3077.203,E2 -3077.203} C_VEL
LIN {X 0,Y 554.155,Z 404.906,A -85,B 0,C 180,E1 -3077.317,E2 -3077.317} C_VEL
LIN {X 0,Y 552.822,Z 397.632,A -85,B 0,C 180,E1 -3077.472,E2 -3077.472} C_VEL
LIN {X 0,Y 553.056,Z 382.483,A -85,B 0,C 180,E1 -3079.438,E2 -3079.438} C_VEL
LIN {X 0,Y 553.468,Z 363.115,A -85,B 0,C 180,E1 -3082.033,E2 -3082.033} C_VEL
LIN {X 0,Y 553.852,Z 344.718,A -85,B 0,C 180,E1 -3084.536,E2 -3084.536} C_VEL
LIN {X 0,Y 552.106,Z 336.469,A -85,B 0,C 180,E1 -3085.797,E2 -3085.797} C_VEL
LIN {X 0,Y 552.069,Z 336.342,A -85,B 0,C 180,E1 -3088.551,E2 -3088.551} C_VEL
LIN {X 0,Y 552.093,Z 336.337,A -85,B 0,C 180,E1 -3091.472,E2 -3091.472} C_VEL
LIN {X 0,Y 552.085,Z 336.343,A -85,B 0,C 180,E1 -3094.163,E2 -3094.163} C_VEL
LIN {X 0,Y 552.047,Z 336.341,A -85,B 0,C 180,E1 -3096.752,E2 -3096.752} C_VEL
LIN {X 0,Y 552.077,Z 336.338,A -85,B 0,C 180,E1 -3099.532,E2 -3099.532} C_VEL
LIN {X 0,Y 552.08,Z 336.336,A -85,B 0,C 180,E1 -3102.43,E2 -3102.43} C_VEL
LIN {X 0,Y 552.064,Z 336.341,A -85,B 0,C 180,E1 -3105.559,E2 -3105.559} C_VEL
LIN {X 0,Y 552.05,Z 336.342,A -85,B 0,C 180,E1 -3108.547,E2 -3108.547} C_VEL
LIN {X 0,Y 552.086,Z 336.335,A -85,B 0,C 180,E1 -3111.408,E2 -3111.408} C_VEL
LIN {X 0,Y 552.058,Z 336.341,A -85,B 0,C 180,E1 -3114.563,E2 -3114.563} C_VEL
LIN {X 0,Y 552.094,Z 336.336,A -85,B 0,C 180,E1 -3117.157,E2 -3117.157} C_VEL
LIN {X 0,Y 552.075,Z 336.336,A -85,B 0,C 180,E1 -3119.957,E2 -3119.957} C_VEL
LIN {X 0,Y 552.122,Z 336.523,A -85,B 0,C 180,E1 -3122.186,E2 -3122.186} C_VEL
LIN {X 0,Y 554.299,Z 346.059,A -85,B 0,C 180,E1 -3123.453,E2 -3123.453} C_VEL
LIN {X 0,Y 554.029,Z 366.423,A -85,B 0,C 180,E1 -3125.872,E2 -3125.872} C_VEL
LIN {X 0,Y 553.547,Z 392.764,A -85,B 0,C 180,E1 -3128.981,E2 -3128.981} C_VEL
LIN {X 0,Y 553.432,Z 398.727,A -85,B 0,C 180,E1 -3129.658,E2 -3129.658} C_VEL
LIN {X 0,Y 555.14,Z 408.123,A -85,B 0,C 180,E1 -3129.864,E2 -3129.864} C_VEL
LIN {X 0,Y 554.464,Z 563.061,A -85,B 0,C 180,E1 -3131.94,E2 -3131.94} C_VEL
LIN {X 0,Y 554.377,Z 575.945,A -85,B 0,C 180,E1 -3132.211,E2 -3132.211} C_VEL
LIN {X 0,Y 554.074,Z 589.592,A -85,B 0,C 180,E1 -3132.61,E2 -3132.61} C_VEL
LIN {X 0,Y 553.821,Z 604.892,A -85,B 0,C 180,E1 -3133.22,E2 -3133.22} C_VEL
LIN {X 0,Y 553.539,Z 617.646,A -85,B 0,C 180,E1 -3133.875,E2 -3133.875} C_VEL
LIN {X 0,Y 553.277,Z 629.479,A -85,B 0,C 180,E1 -3134.608,E2 -3134.608} C_VEL
LIN {X 0,Y 552.998,Z 639.903,A -85,B 0,C 180,E1 -3135.369,E2 -3135.369} C_VEL
LIN {X 0,Y 552.718,Z 649.798,A -85,B 0,C 180,E1 -3136.207,E2 -3136.207} C_VEL
LIN {X 0,Y 552.528,Z 659.268,A -85,B 0,C 180,E1 -3137.138,E2 -3137.138} C_VEL
LIN {X 0,Y 552.28,Z 669.042,A -85,B 0,C 180,E1 -3138.252,E2 -3138.252} C_VEL
LIN {X 0,Y 552.102,Z 679.772,A -85,B 0,C 180,E1 -3139.734,E2 -3139.734} C_VEL
LIN {X 0,Y 551.921,Z 687.46,A -85,B 0,C 180,E1 -3141.026,E2 -3141.026} C_VEL
LIN {X 0,Y 551.839,Z 693.867,A -85,B 0,C 180,E1 -3142.315,E2 -3142.315} C_VEL
LIN {X 0,Y 551.747,Z 699.489,A -85,B 0,C 180,E1 -3143.704,E2 -3143.704} C_VEL
LIN {X 0,Y 551.712,Z 703.266,A -85,B 0,C 180,E1 -3144.884,E2 -3144.884} C_VEL
LIN {X 0,Y 551.73,Z 706.821,A -85,B 0,C 180,E1 -3146.348,E2 -3146.348} C_VEL
LIN {X 0,Y 551.655,Z 709.133,A -85,B 0,C 180,E1 -3147.81,E2 -3147.81} C_VEL
LIN {X 0,Y 551.637,Z 710.287,A -85,B 0,C 180,E1 -3149.27,E2 -3149.27} C_VEL
LIN {X 0,Y 551.638,Z 710.317,A -85,B 0,C 180,E1 -3150.73,E2 -3150.73} C_VEL
LIN {X 0,Y 551.655,Z 709.229,A -85,B 0,C 180,E1 -3152.19,E2 -3152.19} C_VEL
LIN {X 0,Y 551.732,Z 706.998,A -85,B 0,C 180,E1 -3153.652,E2 -3153.652} C_VEL
LIN {X 0,Y 551.785,Z 702.426,A -85,B 0,C 180,E1 -3155.482,E2 -3155.482} C_VEL
LIN {X 0,Y 551.781,Z 698.739,A -85,B 0,C 180,E1 -3156.582,E2 -3156.582} C_VEL
LIN {X 0,Y 551.831,Z 694.281,A -85,B 0,C 180,E1 -3157.685,E2 -3157.685} C_VEL
LIN {X 0,Y 551.917,Z 687.948,A -85,B 0,C 180,E1 -3158.974,E2 -3158.974} C_VEL
LIN {X 0,Y 552.07,Z 681.508,A -85,B 0,C 180,E1 -3160.081,E2 -3160.081} C_VEL
LIN {X 0,Y 552.154,Z 674.146,A -85,B 0,C 180,E1 -3161.165,E2 -3161.165} C_VEL
LIN {X 0,Y 552.379,Z 665.129,A -85,B 0,C 180,E1 -3162.305,E2 -3162.305} C_VEL
LIN {X 0,Y 552.642,Z 654.768,A -85,B 0,C 180,E1 -3163.42,E2 -3163.42} C_VEL
LIN {X 0,Y 552.935,Z 642.217,A -85,B 0,C 180,E1 -3164.538,E2 -3164.538} C_VEL
LIN {X 0,Y 553.237,Z 630.688,A -85,B 0,C 180,E1 -3165.399,E2 -3165.399} C_VEL
LIN {X 0,Y 553.448,Z 620.776,A -85,B 0,C 180,E1 -3166.033,E2 -3166.033} C_VEL
LIN {X 0,Y 553.763,Z 608.615,A -85,B 0,C 180,E1 -3166.687,E2 -3166.687} C_VEL
LIN {X 0,Y 553.963,Z 598.123,A -85,B 0,C 180,E1 -3167.156,E2 -3167.156} C_VEL
LIN {X 0,Y 554.168,Z 585.819,A -85,B 0,C 180,E1 -3167.601,E2 -3167.601} C_VEL
LIN {X 0,Y 554.379,Z 572.828,A -85,B 0,C 180,E1 -3167.957,E2 -3167.957} C_VEL
LIN {X 0,Y 554.529,Z 557.564,A -85,B 0,C 180,E1 -3168.241,E2 -3168.241} C_VEL
LIN {X 0,Y 555.07,Z 407.286,A -85,B 0,C 180,E1 -3170.239,E2 -3170.239} C_VEL
LIN {X 0,Y 553.413,Z 398.62,A -85,B 0,C 180,E1 -3170.439,E2 -3170.439} C_VEL
LIN {X 0,Y 553.883,Z 375.415,A -85,B 0,C 180,E1 -3173.163,E2 -3173.163} C_VEL
LIN {X 0,Y 554.315,Z 349.925,A -85,B 0,C 180,E1 -3176.175,E2 -3176.175} C_VEL
LIN {X 0,Y 554.162,Z 345.108,A -85,B 0,C 180,E1 -3176.758,E2 -3176.758} C_VEL
LIN {X 0,Y 552.088,Z 336.479,A -85,B 0,C 180,E1 -3177.919,E2 -3177.919} C_VEL
LIN {X 0,Y 552.071,Z 336.34,A -85,B 0,C 180,E1 -3180.611,E2 -3180.611} C_VEL
LIN {X 0,Y 552.087,Z 336.336,A -85,B 0,C 180,E1 -3183.188,E2 -3183.188} C_VEL
LIN {X 0,Y 552.062,Z 336.344,A -85,B 0,C 180,E1 -3185.845,E2 -3185.845} C_VEL
LIN {X 0,Y 552.086,Z 336.335,A -85,B 0,C 180,E1 -3188.592,E2 -3188.592} C_VEL
LIN {X 0,Y 552.05,Z 336.343,A -85,B 0,C 180,E1 -3191.452,E2 -3191.452} C_VEL
LIN {X 0,Y 552.074,Z 336.337,A -85,B 0,C 180,E1 -3194.529,E2 -3194.529} C_VEL
LIN {X 0,Y 552.08,Z 336.342,A -85,B 0,C 180,E1 -3197.59,E2 -3197.59} C_VEL
LIN {X 0,Y 552.112,Z 336.33,A -85,B 0,C 180,E1 -3200.94,E2 -3200.94} C_VEL
LIN {X 0,Y 552.095,Z 336.337,A -85,B 0,C 180,E1 -3203.319,E2 -3203.319} C_VEL
LIN {X 0,Y 552.113,Z 336.338,A -85,B 0,C 180,E1 -3205.938,E2 -3205.938} C_VEL
LIN {X 0,Y 552.121,Z 336.328,A -85,B 0,C 180,E1 -3208.541,E2 -3208.541} C_VEL
LIN {X 0,Y 552.095,Z 336.339,A -85,B 0,C 180,E1 -3211.444,E2 -3211.444} C_VEL
LIN {X 0,Y 552.078,Z 336.336,A -85,B 0,C 180,E1 -3214.353,E2 -3214.353} C_VEL
LIN {X 0,Y 552.095,Z 336.333,A -85,B 0,C 180,E1 -3216.758,E2 -3216.758} C_VEL
LIN {X 0,Y 552.117,Z 336.331,A -85,B 0,C 180,E1 -3219.12,E2 -3219.12} C_VEL
LIN {X 0,Y 552.089,Z 336.342,A -85,B 0,C 180,E1 -3221.443,E2 -3221.443} C_VEL
LIN {X 0,Y 552.105,Z 336.338,A -85,B 0,C 180,E1 -3223.737,E2 -3223.737} C_VEL
LIN {X 0,Y 552.133,Z 336.332,A -85,B 0,C 180,E1 -3226.004,E2 -3226.004} C_VEL
LIN {X 0,Y 552.161,Z 336.324,A -85,B 0,C 180,E1 -3228.993,E2 -3228.993} C_VEL
LIN {X 0,Y 552.141,Z 336.331,A -85,B 0,C 180,E1 -3231.951,E2 -3231.951} C_VEL
LIN {X 0,Y 552.223,Z 336.316,A -85,B 0,C 180,E1 -3234.889,E2 -3234.889} C_VEL
LIN {X 0,Y 552.226,Z 336.321,A -85,B 0,C 180,E1 -3237.812,E2 -3237.812} C_VEL
LIN {X 0,Y 552.235,Z 336.315,A -85,B 0,C 180,E1 -3240.729,E2 -3240.729} C_VEL
LIN {X 0,Y 552.198,Z 336.32,A -85,B 0,C 180,E1 -3242.918,E2 -3242.918} C_VEL
LIN {X 0,Y 552.199,Z 336.321,A -85,B 0,C 180,E1 -3245.844,E2 -3245.844} C_VEL
LIN {X 0,Y 552.145,Z 336.325,A -85,B 0,C 180,E1 -3248.786,E2 -3248.786} C_VEL
LIN {X 0,Y 552.164,Z 336.326,A -85,B 0,C 180,E1 -3251.75,E2 -3251.75} C_VEL
LIN {X 0,Y 552.129,Z 336.327,A -85,B 0,C 180,E1 -3254.748,E2 -3254.748} C_VEL
LIN {X 0,Y 552.1,Z 336.333,A -85,B 0,C 180,E1 -3257.789,E2 -3257.789} C_VEL
LIN {X 0,Y 552.127,Z 336.327,A -85,B 0,C 180,E1 -3260.101,E2 -3260.101} C_VEL
LIN {X 0,Y 552.092,Z 336.334,A -85,B 0,C 180,E1 -3262.451,E2 -3262.451} C_VEL
LIN {X 0,Y 552.156,Z 336.332,A -85,B 0,C 180,E1 -3265.35,E2 -3265.35} C_VEL
LIN {X 0,Y 552.11,Z 336.332,A -85,B 0,C 180,E1 -3268.098,E2 -3268.098} C_VEL
LIN {X 0,Y 552.105,Z 336.332,A -85,B 0,C 180,E1 -3270.609,E2 -3270.609} C_VEL
LIN {X 0,Y 552.116,Z 336.337,A -85,B 0,C 180,E1 -3273.186,E2 -3273.186} C_VEL
LIN {X 0,Y 552.086,Z 336.335,A -85,B 0,C 180,E1 -3275.844,E2 -3275.844} C_VEL
LIN {X 0,Y 552.126,Z 336.33,A -85,B 0,C 180,E1 -3279.062,E2 -3279.062} C_VEL
LIN {X 0,Y 552.138,Z 336.329,A -85,B 0,C 180,E1 -3281.444,E2 -3281.444} C_VEL
LIN {X 0,Y 552.096,Z 336.337,A -85,B 0,C 180,E1 -3284.532,E2 -3284.532} C_VEL
LIN {X 0,Y 552.131,Z 336.328,A -85,B 0,C 180,E1 -3287.584,E2 -3287.584} C_VEL
LIN {X 0,Y 552.135,Z 336.332,A -85,B 0,C 180,E1 -3290.473,E2 -3290.473} C_VEL
LIN {X 0,Y 552.107,Z 336.336,A -85,B 0,C 180,E1 -3293.317,E2 -3293.317} C_VEL
LIN {X 0,Y 552.127,Z 336.331,A -85,B 0,C 180,E1 -3295.939,E2 -3295.939} C_VEL
LIN {X 0,Y 552.119,Z 336.336,A -85,B 0,C 180,E1 -3298.541,E2 -3298.541} C_VEL
LIN {X 0,Y 552.125,Z 336.332,A -85,B 0,C 180,E1 -3301.438,E2 -3301.438} C_VEL
LIN {X 0,Y 552.176,Z 336.545,A -85,B 0,C 180,E1 -3302.772,E2 -3302.772} C_VEL
LIN {X 0,Y 554.671,Z 347.034,A -85,B 0,C 180,E1 -3304.107,E2 -3304.107} C_VEL
LIN {X 0,Y 554.08,Z 372.103,A -85,B 0,C 180,E1 -3306.846,E2 -3306.846} C_VEL
LIN {X 0,Y 553.631,Z 397.975,A -85,B 0,C 180,E1 -3309.603,E2 -3309.603} C_VEL
LIN {X 0,Y 555.188,Z 407.778,A -85,B 0,C 180,E1 -3309.817,E2 -3309.817} C_VEL
LIN {X 0,Y 554.471,Z 565.073,A -85,B 0,C 180,E1 -3311.922,E2 -3311.922} C_VEL
LIN {X 0,Y 554.299,Z 580.704,A -85,B 0,C 180,E1 -3312.284,E2 -3312.284} C_VEL
LIN {X 0,Y 554.015,Z 596.037,A -85,B 0,C 180,E1 -3312.799,E2 -3312.799} C_VEL
LIN {X 0,Y 553.791,Z 609.779,A -85,B 0,C 180,E1 -3313.409,E2 -3313.409} C_VEL
LIN {X 0,Y 553.405,Z 623.252,A -85,B 0,C 180,E1 -3314.155,E2 -3314.155} C_VEL
LIN {X 0,Y 553.086,Z 636.287,A -85,B 0,C 180,E1 -3315.04,E2 -3315.04} C_VEL
LIN {X 0,Y 552.78,Z 648.293,A -85,B 0,C 180,E1 -3316.021,E2 -3316.021} C_VEL
LIN {X 0,Y 552.529,Z 659.75,A -85,B 0,C 180,E1 -3317.139,E2 -3317.139} C_VEL
LIN {X 0,Y 552.252,Z 670.438,A -85,B 0,C 180,E1 -3318.383,E2 -3318.383} C_VEL
LIN {X 0,Y 552.124,Z 678.856,A -85,B 0,C 180,E1 -3319.549,E2 -3319.549} C_VEL
LIN {X 0,Y 551.958,Z 686.736,A -85,B 0,C 180,E1 -3320.842,E2 -3320.842} C_VEL
LIN {X 0,Y 551.837,Z 694.091,A -85,B 0,C 180,E1 -3322.315,E2 -3322.315} C_VEL
LIN {X 0,Y 551.769,Z 699.571,A -85,B 0,C 180,E1 -3323.681,E2 -3323.681} C_VEL
LIN {X 0,Y 551.713,Z 703.387,A -85,B 0,C 180,E1 -3324.884,E2 -3324.884} C_VEL
LIN {X 0,Y 551.731,Z 706.889,A -85,B 0,C 180,E1 -3326.348,E2 -3326.348} C_VEL
LIN {X 0,Y 551.654,Z 709.191,A -85,B 0,C 180,E1 -3327.81,E2 -3327.81} C_VEL
LIN {X 0,Y 551.637,Z 710.348,A -85,B 0,C 180,E1 -3329.27,E2 -3329.27} C_VEL
LIN {X 0,Y 551.637,Z 710.348,A -85,B 0,C 180,E1 -3330.73,E2 -3330.73} C_VEL
LIN {X 0,Y 551.654,Z 709.188,A -85,B 0,C 180,E1 -3332.19,E2 -3332.19} C_VEL
LIN {X 0,Y 551.731,Z 706.885,A -85,B 0,C 180,E1 -3333.652,E2 -3333.652} C_VEL
LIN {X 0,Y 551.713,Z 703.386,A -85,B 0,C 180,E1 -3335.116,E2 -3335.116} C_VEL
LIN {X 0,Y 551.78,Z 698.608,A -85,B 0,C 180,E1 -3336.583,E2 -3336.583} C_VEL
LIN {X 0,Y 551.877,Z 692.421,A -85,B 0,C 180,E1 -3338.053,E2 -3338.053} C_VEL
LIN {X 0,Y 551.95,Z 684.644,A -85,B 0,C 180,E1 -3339.528,E2 -3339.528} C_VEL
LIN {X 0,Y 552.183,Z 676.367,A -85,B 0,C 180,E1 -3340.821,E2 -3340.821} C_VEL
LIN {X 0,Y 552.353,Z 666.39,A -85,B 0,C 180,E1 -3342.119,E2 -3342.119} C_VEL
LIN {X 0,Y 552.609,Z 656.185,A -85,B 0,C 180,E1 -3343.234,E2 -3343.234} C_VEL
LIN {X 0,Y 552.889,Z 644.017,A -85,B 0,C 180,E1 -3344.352,E2 -3344.352} C_VEL
LIN {X 0,Y 553.246,Z 631.44,A -85,B 0,C 180,E1 -3345.31,E2 -3345.31} C_VEL
LIN {X 0,Y 553.51,Z 618.505,A -85,B 0,C 180,E1 -3346.126,E2 -3346.126} C_VEL
LIN {X 0,Y 553.827,Z 603.821,A -85,B 0,C 180,E1 -3346.875,E2 -3346.875} C_VEL
LIN {X 0,Y 554.139,Z 589.61,A -85,B 0,C 180,E1 -3347.436,E2 -3347.436} C_VEL
LIN {X 0,Y 554.363,Z 574.3,A -85,B 0,C 180,E1 -3347.882,E2 -3347.882} C_VEL
LIN {X 0,Y 554.517,Z 558.957,A -85,B 0,C 180,E1 -3348.174,E2 -3348.174} C_VEL
LIN {X 0,Y 555.113,Z 406.303,A -85,B 0,C 180,E1 -3350.206,E2 -3350.206} C_VEL
LIN {X 0,Y 553.624,Z 397.87,A -85,B 0,C 180,E1 -3350.405,E2 -3350.405} C_VEL
LIN {X 0,Y 554.098,Z 370.107,A -85,B 0,C 180,E1 -3353.351,E2 -3353.351} C_VEL
LIN {X 0,Y 554.65,Z 346.902,A -85,B 0,C 180,E1 -3355.889,E2 -3355.889} C_VEL
LIN {X 0,Y 552.173,Z 336.467,A -85,B 0,C 180,E1 -3357.229,E2 -3357.229} C_VEL
LIN {X 0,Y 552.118,Z 336.335,A -85,B 0,C 180,E1 -3360.051,E2 -3360.051} C_VEL
LIN {X 0,Y 552.116,Z 336.339,A -85,B 0,C 180,E1 -3362.846,E2 -3362.846} C_VEL
LIN {X 0,Y 552.094,Z 336.338,A -85,B 0,C 180,E1 -3365.442,E2 -3365.442} C_VEL
LIN {X 0,Y 552.098,Z 336.335,A -85,B 0,C 180,E1 -3367.886,E2 -3367.886} C_VEL
LIN {X 0,Y 552.109,Z 336.339,A -85,B 0,C 180,E1 -3370.481,E2 -3370.481} C_VEL
LIN {X 0,Y 552.108,Z 336.334,A -85,B 0,C 180,E1 -3373.424,E2 -3373.424} C_VEL
LIN {X 0,Y 552.108,Z 336.341,A -85,B 0,C 180,E1 -3376.576,E2 -3376.576} C_VEL
LIN {X 0,Y 552.109,Z 336.334,A -85,B 0,C 180,E1 -3379.519,E2 -3379.519} C_VEL
LIN {X 0,Y 552.088,Z 336.343,A -85,B 0,C 180,E1 -3382.336,E2 -3382.336} C_VEL
LIN {X 0,Y 552.077,Z 336.339,A -85,B 0,C 180,E1 -3385.051,E2 -3385.051} C_VEL
LIN {X 0,Y 552.109,Z 336.336,A -85,B 0,C 180,E1 -3387.681,E2 -3387.681} C_VEL
LIN {X 0,Y 552.076,Z 336.345,A -85,B 0,C 180,E1 -3390.233,E2 -3390.233} C_VEL
LIN {X 0,Y 552.076,Z 336.343,A -85,B 0,C 180,E1 -3393.013,E2 -3393.013} C_VEL
LIN {X 0,Y 552.128,Z 336.541,A -85,B 0,C 180,E1 -3394.28,E2 -3394.28} C_VEL
LIN {X 0,Y 553.824,Z 344.199,A -85,B 0,C 180,E1 -3395.443,E2 -3395.443} C_VEL
LIN {X 0,Y 553.759,Z 352.853,A -85,B 0,C 180,E1 -3396.634,E2 -3396.634} C_VEL
LIN {X 0,Y 553.257,Z 374.4,A -85,B 0,C 180,E1 -3399.554,E2 -3399.554} C_VEL
LIN {X 0,Y 552.852,Z 394.451,A -85,B 0,C 180,E1 -3402.236,E2 -3402.236} C_VEL
LIN {X 0,Y 552.847,Z 397.61,A -85,B 0,C 180,E1 -3402.613,E2 -3402.613} C_VEL
LIN {X 0,Y 554.237,Z 406.39,A -85,B 0,C 180,E1 -3402.795,E2 -3402.795} C_VEL
LIN {X 0,Y 553.763,Z 536.059,A -85,B 0,C 180,E1 -3404.519,E2 -3404.519} C_VEL
LIN {X 0,Y 553.611,Z 550.711,A -85,B 0,C 180,E1 -3404.875,E2 -3404.875} C_VEL
LIN {X 0,Y 553.37,Z 563.724,A -85,B 0,C 180,E1 -3405.332,E2 -3405.332} C_VEL
LIN {X 0,Y 553.169,Z 576.78,A -85,B 0,C 180,E1 -3405.937,E2 -3405.937} C_VEL
LIN {X 0,Y 552.9,Z 589.459,A -85,B 0,C 180,E1 -3406.68,E2 -3406.68} C_VEL
LIN {X 0,Y 552.645,Z 600.871,A -85,B 0,C 180,E1 -3407.515,E2 -3407.515} C_VEL
LIN {X 0,Y 552.448,Z 611.027,A -85,B 0,C 180,E1 -3408.397,E2 -3408.397} C_VEL
LIN {X 0,Y 552.26,Z 620.307,A -85,B 0,C 180,E1 -3409.367,E2 -3409.367} C_VEL
LIN {X 0,Y 552.076,Z 629.222,A -85,B 0,C 180,E1 -3410.474,E2 -3410.474} C_VEL
LIN {X 0,Y 551.937,Z 637.753,A -85,B 0,C 180,E1 -3411.764,E2 -3411.764} C_VEL
LIN {X 0,Y 551.822,Z 644.626,A -85,B 0,C 180,E1 -3413.051,E2 -3413.051} C_VEL
LIN {X 0,Y 551.792,Z 650.762,A -85,B 0,C 180,E1 -3414.519,E2 -3414.519} C_VEL
LIN {X 0,Y 551.76,Z 654.29,A -85,B 0,C 180,E1 -3415.617,E2 -3415.617} C_VEL
LIN {X 0,Y 551.72,Z 657.762,A -85,B 0,C 180,E1 -3417.079,E2 -3417.079} C_VEL
LIN {X 0,Y 551.643,Z 659.754,A -85,B 0,C 180,E1 -3418.54,E2 -3418.54} C_VEL
LIN {X 0,Y 551.64,Z 660.496,A -85,B 0,C 180,E1 -3420,E2 -3420} C_VEL
LIN {X 0,Y 551.64,Z 659.834,A -85,B 0,C 180,E1 -3421.46,E2 -3421.46} C_VEL
LIN {X 0,Y 551.719,Z 657.926,A -85,B 0,C 180,E1 -3422.921,E2 -3422.921} C_VEL
LIN {X 0,Y 551.76,Z 654.547,A -85,B 0,C 180,E1 -3424.383,E2 -3424.383} C_VEL
LIN {X 0,Y 551.824,Z 649.765,A -85,B 0,C 180,E1 -3425.848,E2 -3425.848} C_VEL
LIN {X 0,Y 551.824,Z 645.053,A -85,B 0,C 180,E1 -3426.949,E2 -3426.949} C_VEL
LIN {X 0,Y 551.914,Z 638.286,A -85,B 0,C 180,E1 -3428.236,E2 -3428.236} C_VEL
LIN {X 0,Y 552.05,Z 629.863,A -85,B 0,C 180,E1 -3429.526,E2 -3429.526} C_VEL
LIN {X 0,Y 552.233,Z 621.105,A -85,B 0,C 180,E1 -3430.634,E2 -3430.634} C_VEL
LIN {X 0,Y 552.46,Z 610.435,A -85,B 0,C 180,E1 -3431.744,E2 -3431.744} C_VEL
LIN {X 0,Y 552.666,Z 599.717,A -85,B 0,C 180,E1 -3432.672,E2 -3432.672} C_VEL
LIN {X 0,Y 552.9,Z 587.917,A -85,B 0,C 180,E1 -3433.507,E2 -3433.507} C_VEL
LIN {X 0,Y 553.213,Z 574.955,A -85,B 0,C 180,E1 -3434.249,E2 -3434.249} C_VEL
LIN {X 0,Y 553.451,Z 562.641,A -85,B 0,C 180,E1 -3434.8,E2 -3434.8} C_VEL
LIN {X 0,Y 553.61,Z 549.237,A -85,B 0,C 180,E1 -3435.256,E2 -3435.256} C_VEL
LIN {X 0,Y 553.779,Z 535.775,A -85,B 0,C 180,E1 -3435.575,E2 -3435.575} C_VEL
LIN {X 0,Y 554.188,Z 413.402,A -85,B 0,C 180,E1 -3437.203,E2 -3437.203} C_VEL
LIN {X 0,Y 553.601,Z 409.381,A -85,B 0,C 180,E1 -3437.275,E2 -3437.275} C_VEL
LIN {X 0,Y 551.272,Z 404.49,A -85,B 0,C 180,E1 -3437.416,E2 -3437.416} C_VEL
LIN {X 0,Y 546.874,Z 398.089,A -85,B 0,C 180,E1 -3437.717,E2 -3437.717} C_VEL
LIN {X 0,Y 545.939,Z 395.706,A -85,B 0,C 180,E1 -3437.935,E2 -3437.935} C_VEL
LIN {X 0,Y 545.911,Z 395.281,A -85,B 0,C 180,E1 -3437.987,E2 -3437.987} C_VEL
LIN {X 0,Y 546.435,Z 372.079,A -85,B 0,C 180,E1 -3441.108,E2 -3441.108} C_VEL
LIN {X 0,Y 547.036,Z 348.957,A -85,B 0,C 180,E1 -3444.275,E2 -3444.275} C_VEL
LIN {X 0,Y 546.709,Z 344.599,A -85,B 0,C 180,E1 -3444.898,E2 -3444.898} C_VEL
LIN {X 0,Y 545.081,Z 337.481,A -85,B 0,C 180,E1 -3446.001,E2 -3446.001} C_VEL
LIN {X 0,Y 545.015,Z 337.213,A -85,B 0,C 180,E1 -3446.416,E2 -3446.416} C_VEL
LIN {X 0,Y 545.015,Z 337.219,A -85,B 0,C 180,E1 -3449.341,E2 -3449.341} C_VEL
LIN {X 0,Y 545.039,Z 337.221,A -85,B 0,C 180,E1 -3451.916,E2 -3451.916} C_VEL
LIN {X 0,Y 545.04,Z 337.216,A -85,B 0,C 180,E1 -3454.566,E2 -3454.566} C_VEL
LIN {X 0,Y 545.006,Z 337.218,A -85,B 0,C 180,E1 -3457.307,E2 -3457.307} C_VEL
LIN {X 0,Y 545.007,Z 337.225,A -85,B 0,C 180,E1 -3460.148,E2 -3460.148} C_VEL
LIN {X 0,Y 544.999,Z 337.214,A -85,B 0,C 180,E1 -3463.115,E2 -3463.115} C_VEL
LIN {X 0,Y 545.024,Z 337.222,A -85,B 0,C 180,E1 -3465.867,E2 -3465.867} C_VEL
LIN {X 0,Y 544.993,Z 337.219,A -85,B 0,C 180,E1 -3468.877,E2 -3468.877} C_VEL
LIN {X 0,Y 545.027,Z 337.22,A -85,B 0,C 180,E1 -3471.867,E2 -3471.867} C_VEL
LIN {X 0,Y 545.019,Z 337.219,A -85,B 0,C 180,E1 -3474.53,E2 -3474.53} C_VEL
LIN {X 0,Y 545.049,Z 337.214,A -85,B 0,C 180,E1 -3477.21,E2 -3477.21} C_VEL
LIN {X 0,Y 545.024,Z 337.214,A -85,B 0,C 180,E1 -3479.808,E2 -3479.808} C_VEL
LIN {X 0,Y 545.056,Z 337.414,A -85,B 0,C 180,E1 -3481.951,E2 -3481.951} C_VEL
LIN {X 0,Y 547.422,Z 347.399,A -85,B 0,C 180,E1 -3483.298,E2 -3483.298} C_VEL
LIN {X 0,Y 547.293,Z 360.905,A -85,B 0,C 180,E1 -3484.927,E2 -3484.927} C_VEL
LIN {X 0,Y 546.828,Z 383.333,A -85,B 0,C 180,E1 -3487.596,E2 -3487.596} C_VEL
LIN {X 0,Y 546.544,Z 398.472,A -85,B 0,C 180,E1 -3489.38,E2 -3489.38} C_VEL
LIN {X 0,Y 548.478,Z 409.466,A -85,B 0,C 180,E1 -3489.628,E2 -3489.628} C_VEL
LIN {X 0,Y 547.722,Z 563.495,A -85,B 0,C 180,E1 -3491.717,E2 -3491.717} C_VEL
LIN {X 0,Y 547.605,Z 575.574,A -85,B 0,C 180,E1 -3491.974,E2 -3491.974} C_VEL
LIN {X 0,Y 547.373,Z 587.413,A -85,B 0,C 180,E1 -3492.318,E2 -3492.318} C_VEL
LIN {X 0,Y 547.086,Z 599.391,A -85,B 0,C 180,E1 -3492.766,E2 -3492.766} C_VEL
LIN {X 0,Y 546.843,Z 612.509,A -85,B 0,C 180,E1 -3493.384,E2 -3493.384} C_VEL
LIN {X 0,Y 546.445,Z 626.948,A -85,B 0,C 180,E1 -3494.235,E2 -3494.235} C_VEL
LIN {X 0,Y 546.125,Z 638.719,A -85,B 0,C 180,E1 -3495.085,E2 -3495.085} C_VEL
LIN {X 0,Y 545.821,Z 648.768,A -85,B 0,C 180,E1 -3495.934,E2 -3495.934} C_VEL
LIN {X 0,Y 545.576,Z 657.482,A -85,B 0,C 180,E1 -3496.782,E2 -3496.782} C_VEL
LIN {X 0,Y 545.338,Z 665.927,A -85,B 0,C 180,E1 -3497.723,E2 -3497.723} C_VEL
LIN {X 0,Y 545.164,Z 672.868,A -85,B 0,C 180,E1 -3498.603,E2 -3498.603} C_VEL
LIN {X 0,Y 545.035,Z 680.935,A -85,B 0,C 180,E1 -3499.787,E2 -3499.787} C_VEL
LIN {X 0,Y 544.874,Z 687.457,A -85,B 0,C 180,E1 -3500.909,E2 -3500.909} C_VEL
LIN {X 0,Y 544.774,Z 693.862,A -85,B 0,C 180,E1 -3502.215,E2 -3502.215} C_VEL
LIN {X 0,Y 544.656,Z 699.865,A -85,B 0,C 180,E1 -3503.723,E2 -3503.723} C_VEL
LIN {X 0,Y 544.641,Z 703.269,A -85,B 0,C 180,E1 -3504.817,E2 -3504.817} C_VEL
LIN {X 0,Y 544.645,Z 706.825,A -85,B 0,C 180,E1 -3506.301,E2 -3506.301} C_VEL
LIN {X 0,Y 544.569,Z 709.132,A -85,B 0,C 180,E1 -3507.781,E2 -3507.781} C_VEL
LIN {X 0,Y 544.537,Z 710.281,A -85,B 0,C 180,E1 -3509.26,E2 -3509.26} C_VEL
LIN {X 0,Y 544.539,Z 710.496,A -85,B 0,C 180,E1 -3510,E2 -3510} C_VEL
LIN {X 0,Y 544.544,Z 709.954,A -85,B 0,C 180,E1 -3511.479,E2 -3511.479} C_VEL
LIN {X 0,Y 544.645,Z 708.24,A -85,B 0,C 180,E1 -3512.959,E2 -3512.959} C_VEL
LIN {X 0,Y 544.646,Z 707,A -85,B 0,C 180,E1 -3513.699,E2 -3513.699} C_VEL
LIN {X 0,Y 544.713,Z 702.417,A -85,B 0,C 180,E1 -3515.553,E2 -3515.553} C_VEL
LIN {X 0,Y 544.725,Z 697.33,A -85,B 0,C 180,E1 -3517.04,E2 -3517.04} C_VEL
LIN {X 0,Y 544.818,Z 690.862,A -85,B 0,C 180,E1 -3518.531,E2 -3518.531} C_VEL
LIN {X 0,Y 544.981,Z 682.663,A -85,B 0,C 180,E1 -3520.026,E2 -3520.026} C_VEL
LIN {X 0,Y 545.11,Z 675.288,A -85,B 0,C 180,E1 -3521.151,E2 -3521.151} C_VEL
LIN {X 0,Y 545.33,Z 666.67,A -85,B 0,C 180,E1 -3522.277,E2 -3522.277} C_VEL
LIN {X 0,Y 545.571,Z 658.331,A -85,B 0,C 180,E1 -3523.218,E2 -3523.218} C_VEL
LIN {X 0,Y 545.871,Z 647.689,A -85,B 0,C 180,E1 -3524.255,E2 -3524.255} C_VEL
LIN {X 0,Y 546.233,Z 634.717,A -85,B 0,C 180,E1 -3525.318,E2 -3525.318} C_VEL
LIN {X 0,Y 546.549,Z 622.354,A -85,B 0,C 180,E1 -3526.145,E2 -3526.145} C_VEL
LIN {X 0,Y 546.898,Z 610.489,A -85,B 0,C 180,E1 -3526.806,E2 -3526.806} C_VEL
LIN {X 0,Y 547.128,Z 599.243,A -85,B 0,C 180,E1 -3527.328,E2 -3527.328} C_VEL
LIN {X 0,Y 547.372,Z 587.223,A -85,B 0,C 180,E1 -3527.779,E2 -3527.779} C_VEL
LIN {X 0,Y 547.573,Z 575.241,A -85,B 0,C 180,E1 -3528.126,E2 -3528.126} C_VEL
LIN {X 0,Y 547.742,Z 563.532,A -85,B 0,C 180,E1 -3528.371,E2 -3528.371} C_VEL
LIN {X 0,Y 548.459,Z 408.632,A -85,B 0,C 180,E1 -3530.474,E2 -3530.474} C_VEL
LIN {X 0,Y 546.551,Z 398.583,A -85,B 0,C 180,E1 -3530.702,E2 -3530.702} C_VEL
LIN {X 0,Y 547.031,Z 375.119,A -85,B 0,C 180,E1 -3533.47,E2 -3533.47} C_VEL
LIN {X 0,Y 547.487,Z 350.021,A -85,B 0,C 180,E1 -3536.473,E2 -3536.473} C_VEL
LIN {X 0,Y 547.301,Z 346.721,A -85,B 0,C 180,E1 -3536.88,E2 -3536.88} C_VEL
LIN {X 0,Y 545.046,Z 337.366,A -85,B 0,C 180,E1 -3538.154,E2 -3538.154} C_VEL
LIN {X 0,Y 545.033,Z 337.215,A -85,B 0,C 180,E1 -3541.05,E2 -3541.05} C_VEL
LIN {X 0,Y 545.033,Z 337.217,A -85,B 0,C 180,E1 -3543.674,E2 -3543.674} C_VEL
LIN {X 0,Y 544.998,Z 337.221,A -85,B 0,C 180,E1 -3546.384,E2 -3546.384} C_VEL
LIN {X 0,Y 545.032,Z 337.214,A -85,B 0,C 180,E1 -3549.314,E2 -3549.314} C_VEL
LIN {X 0,Y 545.028,Z 337.219,A -85,B 0,C 180,E1 -3552.108,E2 -3552.108} C_VEL
LIN {X 0,Y 545.02,Z 337.215,A -85,B 0,C 180,E1 -3555.172,E2 -3555.172} C_VEL
LIN {X 0,Y 545.029,Z 337.221,A -85,B 0,C 180,E1 -3557.892,E2 -3557.892} C_VEL
LIN {X 0,Y 545.064,Z 337.208,A -85,B 0,C 180,E1 -3560.817,E2 -3560.817} C_VEL
LIN {X 0,Y 545.03,Z 337.222,A -85,B 0,C 180,E1 -3563.619,E2 -3563.619} C_VEL
LIN {X 0,Y 545.055,Z 337.212,A -85,B 0,C 180,E1 -3566.327,E2 -3566.327} C_VEL
LIN {X 0,Y 545.065,Z 337.207,A -85,B 0,C 180,E1 -3568.952,E2 -3568.952} C_VEL
LIN {X 0,Y 545.074,Z 337.215,A -85,B 0,C 180,E1 -3571.506,E2 -3571.506} C_VEL
LIN {X 0,Y 545.033,Z 337.213,A -85,B 0,C 180,E1 -3574.505,E2 -3574.505} C_VEL
LIN {X 0,Y 545.035,Z 337.215,A -85,B 0,C 180,E1 -3577.242,E2 -3577.242} C_VEL
LIN {X 0,Y 545.117,Z 337.203,A -85,B 0,C 180,E1 -3580.415,E2 -3580.415} C_VEL
LIN {X 0,Y 545.056,Z 337.214,A -85,B 0,C 180,E1 -3583.521,E2 -3583.521} C_VEL
LIN {X 0,Y 545.094,Z 337.211,A -85,B 0,C 180,E1 -3585.82,E2 -3585.82} C_VEL
LIN {X 0,Y 545.118,Z 337.2,A -85,B 0,C 180,E1 -3588.849,E2 -3588.849} C_VEL
LIN {X 0,Y 545.093,Z 337.21,A -85,B 0,C 180,E1 -3591.846,E2 -3591.846} C_VEL
LIN {X 0,Y 545.164,Z 337.195,A -85,B 0,C 180,E1 -3594.08,E2 -3594.08} C_VEL
LIN {X 0,Y 545.161,Z 337.199,A -85,B 0,C 180,E1 -3597.044,E2 -3597.044} C_VEL
LIN {X 0,Y 545.203,Z 337.191,A -85,B 0,C 180,E1 -3600,E2 -3600} C_VEL
LIN {X 0,Y 545.166,Z 337.197,A -85,B 0,C 180,E1 -3602.956,E2 -3602.956} C_VEL
LIN {X 0,Y 545.169,Z 337.196,A -85,B 0,C 180,E1 -3605.919,E2 -3605.919} C_VEL
LIN {X 0,Y 545.107,Z 337.203,A -85,B 0,C 180,E1 -3608.9,E2 -3608.9} C_VEL
LIN {X 0,Y 545.136,Z 337.2,A -85,B 0,C 180,E1 -3611.904,E2 -3611.904} C_VEL
LIN {X 0,Y 545.082,Z 337.207,A -85,B 0,C 180,E1 -3614.944,E2 -3614.944} C_VEL
LIN {X 0,Y 545.072,Z 337.207,A -85,B 0,C 180,E1 -3618.026,E2 -3618.026} C_VEL
LIN {X 0,Y 545.093,Z 337.203,A -85,B 0,C 180,E1 -3620.372,E2 -3620.372} C_VEL
LIN {X 0,Y 545.08,Z 337.209,A -85,B 0,C 180,E1 -3623.559,E2 -3623.559} C_VEL
LIN {X 0,Y 545.08,Z 337.207,A -85,B 0,C 180,E1 -3626,E2 -3626} C_VEL
LIN {X 0,Y 545.09,Z 337.21,A -85,B 0,C 180,E1 -3628.748,E2 -3628.748} C_VEL
LIN {X 0,Y 545.058,Z 337.212,A -85,B 0,C 180,E1 -3631.679,E2 -3631.679} C_VEL
LIN {X 0,Y 545.062,Z 337.21,A -85,B 0,C 180,E1 -3634.564,E2 -3634.564} C_VEL
LIN {X 0,Y 545.038,Z 337.217,A -85,B 0,C 180,E1 -3637.304,E2 -3637.304} C_VEL
LIN {X 0,Y 545.072,Z 337.198,A -85,B 0,C 180,E1 -3640.142,E2 -3640.142} C_VEL
LIN {X 0,Y 545.063,Z 337.212,A -85,B 0,C 180,E1 -3642.697,E2 -3642.697} C_VEL
LIN {X 0,Y 545.063,Z 337.211,A -85,B 0,C 180,E1 -3645.167,E2 -3645.167} C_VEL
LIN {X 0,Y 545.083,Z 337.205,A -85,B 0,C 180,E1 -3647.898,E2 -3647.898} C_VEL
LIN {X 0,Y 545.085,Z 337.215,A -85,B 0,C 180,E1 -3650.819,E2 -3650.819} C_VEL
LIN {X 0,Y 545.042,Z 337.214,A -85,B 0,C 180,E1 -3653.62,E2 -3653.62} C_VEL
LIN {X 0,Y 545.066,Z 337.213,A -85,B 0,C 180,E1 -3656.328,E2 -3656.328} C_VEL
LIN {X 0,Y 545.068,Z 337.217,A -85,B 0,C 180,E1 -3658.952,E2 -3658.952} C_VEL
LIN {X 0,Y 545.101,Z 337.207,A -85,B 0,C 180,E1 -3661.508,E2 -3661.508} C_VEL
LIN {X 0,Y 545.143,Z 337.405,A -85,B 0,C 180,E1 -3662.498,E2 -3662.498} C_VEL
LIN {X 0,Y 547.926,Z 348.776,A -85,B 0,C 180,E1 -3663.969,E2 -3663.969} C_VEL
LIN {X 0,Y 547.227,Z 375.625,A -85,B 0,C 180,E1 -3666.939,E2 -3666.939} C_VEL
LIN {X 0,Y 546.74,Z 397.942,A -85,B 0,C 180,E1 -3669.348,E2 -3669.348} C_VEL
LIN {X 0,Y 548.503,Z 408.224,A -85,B 0,C 180,E1 -3669.577,E2 -3669.577} C_VEL
LIN {X 0,Y 547.724,Z 565.063,A -85,B 0,C 180,E1 -3671.691,E2 -3671.691} C_VEL
LIN {X 0,Y 547.528,Z 580.703,A -85,B 0,C 180,E1 -3672.058,E2 -3672.058} C_VEL
LIN {X 0,Y 547.233,Z 596.034,A -85,B 0,C 180,E1 -3672.579,E2 -3672.579} C_VEL
LIN {X 0,Y 546.965,Z 609.782,A -85,B 0,C 180,E1 -3673.196,E2 -3673.196} C_VEL
LIN {X 0,Y 546.529,Z 623.255,A -85,B 0,C 180,E1 -3673.95,E2 -3673.95} C_VEL
LIN {X 0,Y 546.151,Z 637.128,A -85,B 0,C 180,E1 -3674.908,E2 -3674.908} C_VEL
LIN {X 0,Y 545.818,Z 649.355,A -85,B 0,C 180,E1 -3675.934,E2 -3675.934} C_VEL
LIN {X 0,Y 545.511,Z 661.509,A -85,B 0,C 180,E1 -3677.16,E2 -3677.16} C_VEL
LIN {X 0,Y 545.175,Z 672.105,A -85,B 0,C 180,E1 -3678.446,E2 -3678.446} C_VEL
LIN {X 0,Y 545.05,Z 681.296,A -85,B 0,C 180,E1 -3679.788,E2 -3679.788} C_VEL
LIN {X 0,Y 544.845,Z 688.75,A -85,B 0,C 180,E1 -3681.096,E2 -3681.096} C_VEL
LIN {X 0,Y 544.745,Z 695.701,A -85,B 0,C 180,E1 -3682.587,E2 -3682.587} C_VEL
LIN {X 0,Y 544.709,Z 701.163,A -85,B 0,C 180,E1 -3684.076,E2 -3684.076} C_VEL
LIN {X 0,Y 544.606,Z 705.292,A -85,B 0,C 180,E1 -3685.559,E2 -3685.559} C_VEL
LIN {X 0,Y 544.643,Z 708.185,A -85,B 0,C 180,E1 -3687.041,E2 -3687.041} C_VEL
LIN {X 0,Y 544.543,Z 709.91,A -85,B 0,C 180,E1 -3688.521,E2 -3688.521} C_VEL
LIN {X 0,Y 544.538,Z 710.5,A -85,B 0,C 180,E1 -3690,E2 -3690} C_VEL
LIN {X 0,Y 544.543,Z 709.908,A -85,B 0,C 180,E1 -3691.479,E2 -3691.479} C_VEL
LIN {X 0,Y 544.644,Z 708.181,A -85,B 0,C 180,E1 -3692.959,E2 -3692.959} C_VEL
LIN {X 0,Y 544.606,Z 705.289,A -85,B 0,C 180,E1 -3694.441,E2 -3694.441} C_VEL
LIN {X 0,Y 544.707,Z 701.165,A -85,B 0,C 180,E1 -3695.925,E2 -3695.925} C_VEL
LIN {X 0,Y 544.745,Z 695.701,A -85,B 0,C 180,E1 -3697.413,E2 -3697.413} C_VEL
LIN {X 0,Y 544.845,Z 688.744,A -85,B 0,C 180,E1 -3698.905,E2 -3698.905} C_VEL
LIN {X 0,Y 545.074,Z 680.082,A -85,B 0,C 180,E1 -3700.4,E2 -3700.4} C_VEL
LIN {X 0,Y 545.237,Z 670.706,A -85,B 0,C 180,E1 -3701.735,E2 -3701.735} C_VEL
LIN {X 0,Y 545.511,Z 661.507,A -85,B 0,C 180,E1 -3702.841,E2 -3702.841} C_VEL
LIN {X 0,Y 545.791,Z 649.357,A -85,B 0,C 180,E1 -3704.067,E2 -3704.067} C_VEL
LIN {X 0,Y 546.193,Z 636.805,A -85,B 0,C 180,E1 -3705.115,E2 -3705.115} C_VEL
LIN {X 0,Y 546.529,Z 623.25,A -85,B 0,C 180,E1 -3706.05,E2 -3706.05} C_VEL
LIN {X 0,Y 546.948,Z 609.77,A -85,B 0,C 180,E1 -3706.805,E2 -3706.805} C_VEL
LIN {X 0,Y 547.212,Z 596.039,A -85,B 0,C 180,E1 -3707.422,E2 -3707.422} C_VEL
LIN {X 0,Y 547.537,Z 581.485,A -85,B 0,C 180,E1 -3707.918,E2 -3707.918} C_VEL
LIN {X 0,Y 547.717,Z 566.389,A -85,B 0,C 180,E1 -3708.282,E2 -3708.282} C_VEL
LIN {X 0,Y 547.91,Z 529.735,A -85,B 0,C 180,E1 -3708.801,E2 -3708.801} C_VEL
LIN {X 0,Y 548.378,Z 407.266,A -85,B 0,C 180,E1 -3710.434,E2 -3710.434} C_VEL
LIN {X 0,Y 546.733,Z 397.911,A -85,B 0,C 180,E1 -3710.646,E2 -3710.646} C_VEL
LIN {X 0,Y 547.211,Z 373.557,A -85,B 0,C 180,E1 -3713.262,E2 -3713.262} C_VEL
LIN {X 0,Y 547.894,Z 348.684,A -85,B 0,C 180,E1 -3716.017,E2 -3716.017} C_VEL
LIN {X 0,Y 545.104,Z 337.35,A -85,B 0,C 180,E1 -3717.504,E2 -3717.504} C_VEL
LIN {X 0,Y 545.079,Z 337.213,A -85,B 0,C 180,E1 -3720.246,E2 -3720.246} C_VEL
LIN {X 0,Y 545.08,Z 337.216,A -85,B 0,C 180,E1 -3723.062,E2 -3723.062} C_VEL
LIN {X 0,Y 545.05,Z 337.214,A -85,B 0,C 180,E1 -3725.675,E2 -3725.675} C_VEL
LIN {X 0,Y 545.053,Z 337.215,A -85,B 0,C 180,E1 -3728.237,E2 -3728.237} C_VEL
LIN {X 0,Y 545.082,Z 337.214,A -85,B 0,C 180,E1 -3730.473,E2 -3730.473} C_VEL
LIN {X 0,Y 545.079,Z 337.213,A -85,B 0,C 180,E1 -3733.107,E2 -3733.107} C_VEL
LIN {X 0,Y 545.05,Z 337.217,A -85,B 0,C 180,E1 -3736.226,E2 -3736.226} C_VEL
LIN {X 0,Y 545.081,Z 337.213,A -85,B 0,C 180,E1 -3738.885,E2 -3738.885} C_VEL
LIN {X 0,Y 545.078,Z 337.214,A -85,B 0,C 180,E1 -3740.818,E2 -3740.818} C_VEL
LIN {X 0,Y 545.033,Z 337.216,A -85,B 0,C 180,E1 -3743.619,E2 -3743.619} C_VEL
LIN {X 0,Y 545.063,Z 337.219,A -85,B 0,C 180,E1 -3746.328,E2 -3746.328} C_VEL
LIN {X 0,Y 545.062,Z 337.214,A -85,B 0,C 180,E1 -3748.952,E2 -3748.952} C_VEL
LIN {X 0,Y 545.032,Z 337.219,A -85,B 0,C 180,E1 -3751.504,E2 -3751.504} C_VEL
LIN {X 0,Y 545.092,Z 337.41,A -85,B 0,C 180,E1 -3754.016,E2 -3754.016} C_VEL
LIN {X 0,Y 547.126,Z 347.209,A -85,B 0,C 180,E1 -3755.527,E2 -3755.527} C_VEL
LIN {X 0,Y 546.571,Z 367.388,A -85,B 0,C 180,E1 -3758.304,E2 -3758.304} C_VEL
LIN {X 0,Y 546.099,Z 388.939,A -85,B 0,C 180,E1 -3761.232,E2 -3761.232} C_VEL
LIN {X 0,Y 545.915,Z 397.569,A -85,B 0,C 180,E1 -3762.362,E2 -3762.362} C_VEL
LIN {X 0,Y 547.47,Z 406.674,A -85,B 0,C 180,E1 -3762.573,E2 -3762.573} C_VEL
LIN {X 0,Y 546.933,Z 536.09,A -85,B 0,C 180,E1 -3764.321,E2 -3764.321} C_VEL
LIN {X 0,Y 546.693,Z 550.565,A -85,B 0,C 180,E1 -3764.674,E2 -3764.674} C_VEL
LIN {X 0,Y 546.507,Z 563.73,A -85,B 0,C 180,E1 -3765.144,E2 -3765.144} C_VEL
LIN {X 0,Y 546.254,Z 576.786,A -85,B 0,C 180,E1 -3765.756,E2 -3765.756} C_VEL
LIN {X 0,Y 545.951,Z 589.465,A -85,B 0,C 180,E1 -3766.507,E2 -3766.507} C_VEL
LIN {X 0,Y 545.677,Z 600.872,A -85,B 0,C 180,E1 -3767.353,E2 -3767.353} C_VEL
LIN {X 0,Y 545.427,Z 611.789,A -85,B 0,C 180,E1 -3768.318,E2 -3768.318} C_VEL
LIN {X 0,Y 545.223,Z 621.89,A -85,B 0,C 180,E1 -3769.416,E2 -3769.416} C_VEL
LIN {X 0,Y 545.038,Z 630.598,A -85,B 0,C 180,E1 -3770.537,E2 -3770.537} C_VEL
LIN {X 0,Y 544.854,Z 638.81,A -85,B 0,C 180,E1 -3771.843,E2 -3771.843} C_VEL
LIN {X 0,Y 544.755,Z 646.346,A -85,B 0,C 180,E1 -3773.332,E2 -3773.332} C_VEL
LIN {X 0,Y 544.724,Z 650.759,A -85,B 0,C 180,E1 -3774.447,E2 -3774.447} C_VEL
LIN {X 0,Y 544.654,Z 654.288,A -85,B 0,C 180,E1 -3775.56,E2 -3775.56} C_VEL
LIN {X 0,Y 544.647,Z 657.766,A -85,B 0,C 180,E1 -3777.041,E2 -3777.041} C_VEL
LIN {X 0,Y 544.544,Z 659.749,A -85,B 0,C 180,E1 -3778.521,E2 -3778.521} C_VEL
LIN {X 0,Y 544.54,Z 660.496,A -85,B 0,C 180,E1 -3780,E2 -3780} C_VEL
LIN {X 0,Y 544.542,Z 659.828,A -85,B 0,C 180,E1 -3781.479,E2 -3781.479} C_VEL
LIN {X 0,Y 544.646,Z 657.924,A -85,B 0,C 180,E1 -3782.959,E2 -3782.959} C_VEL
LIN {X 0,Y 544.654,Z 654.541,A -85,B 0,C 180,E1 -3784.44,E2 -3784.44} C_VEL
LIN {X 0,Y 544.741,Z 649.766,A -85,B 0,C 180,E1 -3785.924,E2 -3785.924} C_VEL
LIN {X 0,Y 544.737,Z 645.046,A -85,B 0,C 180,E1 -3787.04,E2 -3787.04} C_VEL
LIN {X 0,Y 544.867,Z 638.277,A -85,B 0,C 180,E1 -3788.344,E2 -3788.344} C_VEL
LIN {X 0,Y 544.993,Z 629.855,A -85,B 0,C 180,E1 -3789.651,E2 -3789.651} C_VEL
LIN {X 0,Y 545.22,Z 621.093,A -85,B 0,C 180,E1 -3790.772,E2 -3790.772} C_VEL
LIN {X 0,Y 545.45,Z 610.421,A -85,B 0,C 180,E1 -3791.897,E2 -3791.897} C_VEL
LIN {X 0,Y 545.72,Z 599.702,A -85,B 0,C 180,E1 -3792.836,E2 -3792.836} C_VEL
LIN {X 0,Y 545.979,Z 587.899,A -85,B 0,C 180,E1 -3793.682,E2 -3793.682} C_VEL
LIN {X 0,Y 546.32,Z 574.935,A -85,B 0,C 180,E1 -3794.433,E2 -3794.433} C_VEL
LIN {X 0,Y 546.58,Z 562.832,A -85,B 0,C 180,E1 -3794.981,E2 -3794.981} C_VEL
LIN {X 0,Y 546.745,Z 549.531,A -85,B 0,C 180,E1 -3795.442,E2 -3795.442} C_VEL
LIN {X 0,Y 546.942,Z 535.719,A -85,B 0,C 180,E1 -3795.774,E2 -3795.774} C_VEL
LIN {X 0,Y 547.437,Z 406.126,A -85,B 0,C 180,E1 -3797.522,E2 -3797.522} C_VEL
LIN {X 0,Y 545.916,Z 397.437,A -85,B 0,C 180,E1 -3797.72,E2 -3797.72} C_VEL
LIN {X 0,Y 545.911,Z 395.281,A -85,B 0,C 180,E1 -3797.987,E2 -3797.987} C_VEL
LIN {X 0,Y 545.313,Z 391.766,A -85,B 0,C 180,E1 -3798.48,E2 -3798.48} C_VEL
LIN {X 0,Y 539.938,Z 381.001,A -85,B 0,C 180,E1 -3800.151,E2 -3800.151} C_VEL
LIN {X 0,Y 539.417,Z 377.489,A -85,B 0,C 180,E1 -3800.655,E2 -3800.655} C_VEL
LIN {X 0,Y 540.062,Z 354.794,A -85,B 0,C 180,E1 -3803.792,E2 -3803.792} C_VEL
LIN {X 0,Y 540.087,Z 347.529,A -85,B 0,C 180,E1 -3804.813,E2 -3804.813} C_VEL
LIN {X 0,Y 538.014,Z 338.245,A -85,B 0,C 180,E1 -3806.283,E2 -3806.283} C_VEL
LIN {X 0,Y 537.974,Z 338.096,A -85,B 0,C 180,E1 -3808.922,E2 -3808.922} C_VEL
LIN {X 0,Y 537.995,Z 338.098,A -85,B 0,C 180,E1 -3811.884,E2 -3811.884} C_VEL
LIN {X 0,Y 537.991,Z 338.094,A -85,B 0,C 180,E1 -3814.614,E2 -3814.614} C_VEL
LIN {X 0,Y 537.97,Z 338.101,A -85,B 0,C 180,E1 -3817.88,E2 -3817.88} C_VEL
LIN {X 0,Y 537.951,Z 338.096,A -85,B 0,C 180,E1 -3820.785,E2 -3820.785} C_VEL
LIN {X 0,Y 537.977,Z 338.094,A -85,B 0,C 180,E1 -3823.819,E2 -3823.819} C_VEL
LIN {X 0,Y 537.977,Z 338.095,A -85,B 0,C 180,E1 -3826.181,E2 -3826.181} C_VEL
LIN {X 0,Y 537.952,Z 338.097,A -85,B 0,C 180,E1 -3829.265,E2 -3829.265} C_VEL
LIN {X 0,Y 537.969,Z 338.101,A -85,B 0,C 180,E1 -3832.12,E2 -3832.12} C_VEL
LIN {X 0,Y 537.99,Z 338.093,A -85,B 0,C 180,E1 -3835.386,E2 -3835.386} C_VEL
LIN {X 0,Y 537.994,Z 338.098,A -85,B 0,C 180,E1 -3838.116,E2 -3838.116} C_VEL
LIN {X 0,Y 537.985,Z 338.096,A -85,B 0,C 180,E1 -3841.095,E2 -3841.095} C_VEL
LIN {X 0,Y 538.025,Z 338.371,A -85,B 0,C 180,E1 -3841.724,E2 -3841.724} C_VEL
LIN {X 0,Y 540.523,Z 348.759,A -85,B 0,C 180,E1 -3843.139,E2 -3843.139} C_VEL
LIN {X 0,Y 540.621,Z 356.032,A -85,B 0,C 180,E1 -3844.036,E2 -3844.036} C_VEL
LIN {X 0,Y 540.034,Z 380.81,A -85,B 0,C 180,E1 -3847.019,E2 -3847.019} C_VEL
LIN {X 0,Y 539.718,Z 398.648,A -85,B 0,C 180,E1 -3849.122,E2 -3849.122} C_VEL
LIN {X 0,Y 541.837,Z 410.284,A -85,B 0,C 180,E1 -3849.38,E2 -3849.38} C_VEL
LIN {X 0,Y 540.999,Z 564.095,A -85,B 0,C 180,E1 -3851.49,E2 -3851.49} C_VEL
LIN {X 0,Y 540.783,Z 579.056,A -85,B 0,C 180,E1 -3851.826,E2 -3851.826} C_VEL
LIN {X 0,Y 540.462,Z 594.821,A -85,B 0,C 180,E1 -3852.353,E2 -3852.353} C_VEL
LIN {X 0,Y 540.167,Z 606.811,A -85,B 0,C 180,E1 -3852.88,E2 -3852.88} C_VEL
LIN {X 0,Y 539.875,Z 617.646,A -85,B 0,C 180,E1 -3853.455,E2 -3853.455} C_VEL
LIN {X 0,Y 539.521,Z 628.312,A -85,B 0,C 180,E1 -3854.124,E2 -3854.124} C_VEL
LIN {X 0,Y 539.214,Z 638.715,A -85,B 0,C 180,E1 -3854.89,E2 -3854.89} C_VEL
LIN {X 0,Y 538.896,Z 648.763,A -85,B 0,C 180,E1 -3855.75,E2 -3855.75} C_VEL
LIN {X 0,Y 538.611,Z 657.48,A -85,B 0,C 180,E1 -3856.608,E2 -3856.608} C_VEL
LIN {X 0,Y 538.333,Z 665.922,A -85,B 0,C 180,E1 -3857.56,E2 -3857.56} C_VEL
LIN {X 0,Y 538.131,Z 673.426,A -85,B 0,C 180,E1 -3858.531,E2 -3858.531} C_VEL
LIN {X 0,Y 538.01,Z 680.93,A -85,B 0,C 180,E1 -3859.653,E2 -3859.653} C_VEL
LIN {X 0,Y 537.83,Z 687.454,A -85,B 0,C 180,E1 -3860.789,E2 -3860.789} C_VEL
LIN {X 0,Y 537.736,Z 692.167,A -85,B 0,C 180,E1 -3861.734,E2 -3861.734} C_VEL
LIN {X 0,Y 537.651,Z 696.987,A -85,B 0,C 180,E1 -3862.866,E2 -3862.866} C_VEL
LIN {X 0,Y 537.641,Z 702.138,A -85,B 0,C 180,E1 -3864.374,E2 -3864.374} C_VEL
LIN {X 0,Y 537.562,Z 706.829,A -85,B 0,C 180,E1 -3866.252,E2 -3866.252} C_VEL
LIN {X 0,Y 537.488,Z 709.13,A -85,B 0,C 180,E1 -3867.752,E2 -3867.752} C_VEL
LIN {X 0,Y 537.437,Z 710.275,A -85,B 0,C 180,E1 -3869.251,E2 -3869.251} C_VEL
LIN {X 0,Y 537.44,Z 710.496,A -85,B 0,C 180,E1 -3870,E2 -3870} C_VEL
LIN {X 0,Y 537.449,Z 709.948,A -85,B 0,C 180,E1 -3871.499,E2 -3871.499} C_VEL
LIN {X 0,Y 537.545,Z 708.232,A -85,B 0,C 180,E1 -3872.998,E2 -3872.998} C_VEL
LIN {X 0,Y 537.563,Z 707.001,A -85,B 0,C 180,E1 -3873.748,E2 -3873.748} C_VEL
LIN {X 0,Y 537.64,Z 702.409,A -85,B 0,C 180,E1 -3875.626,E2 -3875.626} C_VEL
LIN {X 0,Y 537.619,Z 698.724,A -85,B 0,C 180,E1 -3876.757,E2 -3876.757} C_VEL
LIN {X 0,Y 537.695,Z 694.261,A -85,B 0,C 180,E1 -3877.888,E2 -3877.888} C_VEL
LIN {X 0,Y 537.801,Z 687.93,A -85,B 0,C 180,E1 -3879.212,E2 -3879.212} C_VEL
LIN {X 0,Y 537.996,Z 681.483,A -85,B 0,C 180,E1 -3880.348,E2 -3880.348} C_VEL
LIN {X 0,Y 538.122,Z 674.097,A -85,B 0,C 180,E1 -3881.464,E2 -3881.464} C_VEL
LIN {X 0,Y 538.323,Z 666.655,A -85,B 0,C 180,E1 -3882.44,E2 -3882.44} C_VEL
LIN {X 0,Y 538.591,Z 658.318,A -85,B 0,C 180,E1 -3883.392,E2 -3883.392} C_VEL
LIN {X 0,Y 538.881,Z 648.697,A -85,B 0,C 180,E1 -3884.347,E2 -3884.347} C_VEL
LIN {X 0,Y 539.199,Z 638.411,A -85,B 0,C 180,E1 -3885.226,E2 -3885.226} C_VEL
LIN {X 0,Y 539.637,Z 625.468,A -85,B 0,C 180,E1 -3886.163,E2 -3886.163} C_VEL
LIN {X 0,Y 540.019,Z 612.372,A -85,B 0,C 180,E1 -3886.929,E2 -3886.929} C_VEL
LIN {X 0,Y 540.315,Z 600.41,A -85,B 0,C 180,E1 -3887.505,E2 -3887.505} C_VEL
LIN {X 0,Y 540.61,Z 587.229,A -85,B 0,C 180,E1 -3888.009,E2 -3888.009} C_VEL
LIN {X 0,Y 540.908,Z 573.463,A -85,B 0,C 180,E1 -3888.404,E2 -3888.404} C_VEL
LIN {X 0,Y 541.059,Z 558.97,A -85,B 0,C 180,E1 -3888.688,E2 -3888.688} C_VEL
LIN {X 0,Y 541.848,Z 410,A -85,B 0,C 180,E1 -3890.714,E2 -3890.714} C_VEL
LIN {X 0,Y 539.688,Z 398.355,A -85,B 0,C 180,E1 -3890.986,E2 -3890.986} C_VEL
LIN {X 0,Y 540.207,Z 374.846,A -85,B 0,C 180,E1 -3893.785,E2 -3893.785} C_VEL
LIN {X 0,Y 540.669,Z 351.202,A -85,B 0,C 180,E1 -3896.644,E2 -3896.644} C_VEL
LIN {X 0,Y 540.308,Z 347.783,A -85,B 0,C 180,E1 -3897.082,E2 -3897.082} C_VEL
LIN {X 0,Y 538.024,Z 338.251,A -85,B 0,C 180,E1 -3898.396,E2 -3898.396} C_VEL
LIN {X 0,Y 537.988,Z 338.094,A -85,B 0,C 180,E1 -3901.503,E2 -3901.503} C_VEL
LIN {X 0,Y 537.989,Z 338.099,A -85,B 0,C 180,E1 -3904.175,E2 -3904.175} C_VEL
LIN {X 0,Y 537.958,Z 338.096,A -85,B 0,C 180,E1 -3907.163,E2 -3907.163} C_VEL
LIN {X 0,Y 537.968,Z 338.096,A -85,B 0,C 180,E1 -3909.802,E2 -3909.802} C_VEL
LIN {X 0,Y 537.969,Z 338.093,A -85,B 0,C 180,E1 -3912.791,E2 -3912.791} C_VEL
LIN {X 0,Y 537.993,Z 338.091,A -85,B 0,C 180,E1 -3915.136,E2 -3915.136} C_VEL
LIN {X 0,Y 537.979,Z 338.097,A -85,B 0,C 180,E1 -3918.222,E2 -3918.222} C_VEL
LIN {X 0,Y 538.001,Z 338.089,A -85,B 0,C 180,E1 -3921.168,E2 -3921.168} C_VEL
LIN {X 0,Y 537.968,Z 338.096,A -85,B 0,C 180,E1 -3924.093,E2 -3924.093} C_VEL
LIN {X 0,Y 538.031,Z 338.086,A -85,B 0,C 180,E1 -3926.727,E2 -3926.727} C_VEL
LIN {X 0,Y 538.014,Z 338.092,A -85,B 0,C 180,E1 -3929.559,E2 -3929.559} C_VEL
LIN {X 0,Y 538.01,Z 338.09,A -85,B 0,C 180,E1 -3931.948,E2 -3931.948} C_VEL
LIN {X 0,Y 538.014,Z 338.088,A -85,B 0,C 180,E1 -3934.464,E2 -3934.464} C_VEL
LIN {X 0,Y 538.012,Z 338.087,A -85,B 0,C 180,E1 -3936.928,E2 -3936.928} C_VEL
LIN {X 0,Y 538.081,Z 338.081,A -85,B 0,C 180,E1 -3940.148,E2 -3940.148} C_VEL
LIN {X 0,Y 538.003,Z 338.091,A -85,B 0,C 180,E1 -3943.298,E2 -3943.298} C_VEL
LIN {X 0,Y 538.064,Z 338.09,A -85,B 0,C 180,E1 -3945.631,E2 -3945.631} C_VEL
LIN {X 0,Y 538.077,Z 338.076,A -85,B 0,C 180,E1 -3948.701,E2 -3948.701} C_VEL
LIN {X 0,Y 538.059,Z 338.088,A -85,B 0,C 180,E1 -3951.739,E2 -3951.739} C_VEL
LIN {X 0,Y 538.119,Z 338.073,A -85,B 0,C 180,E1 -3954.003,E2 -3954.003} C_VEL
LIN {X 0,Y 538.127,Z 338.074,A -85,B 0,C 180,E1 -3957.005,E2 -3957.005} C_VEL
LIN {X 0,Y 538.174,Z 338.067,A -85,B 0,C 180,E1 -3960,E2 -3960} C_VEL
LIN {X 0,Y 538.133,Z 338.073,A -85,B 0,C 180,E1 -3962.994,E2 -3962.994} C_VEL
LIN {X 0,Y 538.119,Z 338.074,A -85,B 0,C 180,E1 -3965.997,E2 -3965.997} C_VEL
LIN {X 0,Y 538.061,Z 338.082,A -85,B 0,C 180,E1 -3969.018,E2 -3969.018} C_VEL
LIN {X 0,Y 538.084,Z 338.077,A -85,B 0,C 180,E1 -3972.062,E2 -3972.062} C_VEL
LIN {X 0,Y 538.043,Z 338.087,A -85,B 0,C 180,E1 -3975.144,E2 -3975.144} C_VEL
LIN {X 0,Y 538.026,Z 338.084,A -85,B 0,C 180,E1 -3978.27,E2 -3978.27} C_VEL
LIN {X 0,Y 538.038,Z 338.083,A -85,B 0,C 180,E1 -3980.651,E2 -3980.651} C_VEL
LIN {X 0,Y 538.003,Z 338.088,A -85,B 0,C 180,E1 -3983.888,E2 -3983.888} C_VEL
LIN {X 0,Y 538.042,Z 338.083,A -85,B 0,C 180,E1 -3986.367,E2 -3986.367} C_VEL
LIN {X 0,Y 538.031,Z 338.092,A -85,B 0,C 180,E1 -3988.933,E2 -3988.933} C_VEL
LIN {X 0,Y 538.011,Z 338.089,A -85,B 0,C 180,E1 -3991.887,E2 -3991.887} C_VEL
LIN {X 0,Y 538.012,Z 338.088,A -85,B 0,C 180,E1 -3994.618,E2 -3994.618} C_VEL
LIN {X 0,Y 538.005,Z 338.095,A -85,B 0,C 180,E1 -3997.17,E2 -3997.17} C_VEL
LIN {X 0,Y 538.028,Z 338.075,A -85,B 0,C 180,E1 -3999.796,E2 -3999.796} C_VEL
LIN {X 0,Y 538.02,Z 338.09,A -85,B 0,C 180,E1 -4002.786,E2 -4002.786} C_VEL
LIN {X 0,Y 538.032,Z 338.087,A -85,B 0,C 180,E1 -4005.141,E2 -4005.141} C_VEL
LIN {X 0,Y 538.04,Z 338.083,A -85,B 0,C 180,E1 -4008.228,E2 -4008.228} C_VEL
LIN {X 0,Y 538.016,Z 338.094,A -85,B 0,C 180,E1 -4011.17,E2 -4011.17} C_VEL
LIN {X 0,Y 537.994,Z 338.091,A -85,B 0,C 180,E1 -4014.089,E2 -4014.089} C_VEL
LIN {X 0,Y 538.03,Z 338.093,A -85,B 0,C 180,E1 -4016.727,E2 -4016.727} C_VEL
LIN {X 0,Y 538.027,Z 338.092,A -85,B 0,C 180,E1 -4019.556,E2 -4019.556} C_VEL
LIN {X 0,Y 538.062,Z 338.23,A -85,B 0,C 180,E1 -4022.201,E2 -4022.201} C_VEL
LIN {X 0,Y 541.142,Z 350.261,A -85,B 0,C 180,E1 -4023.796,E2 -4023.796} C_VEL
LIN {X 0,Y 540.527,Z 371.91,A -85,B 0,C 180,E1 -4026.23,E2 -4026.23} C_VEL
LIN {X 0,Y 539.897,Z 398.038,A -85,B 0,C 180,E1 -4029.099,E2 -4029.099} C_VEL
LIN {X 0,Y 541.799,Z 409.26,A -85,B 0,C 180,E1 -4029.347,E2 -4029.347} C_VEL
LIN {X 0,Y 540.929,Z 565.195,A -85,B 0,C 180,E1 -4031.479,E2 -4031.479} C_VEL
LIN {X 0,Y 540.731,Z 580.852,A -85,B 0,C 180,E1 -4031.849,E2 -4031.849} C_VEL
LIN {X 0,Y 540.431,Z 595.703,A -85,B 0,C 180,E1 -4032.352,E2 -4032.352} C_VEL
LIN {X 0,Y 540.127,Z 609.681,A -85,B 0,C 180,E1 -4032.977,E2 -4032.977} C_VEL
LIN {X 0,Y 539.671,Z 623.253,A -85,B 0,C 180,E1 -4033.741,E2 -4033.741} C_VEL
LIN {X 0,Y 539.322,Z 636.234,A -85,B 0,C 180,E1 -4034.645,E2 -4034.645} C_VEL
LIN {X 0,Y 538.893,Z 648.289,A -85,B 0,C 180,E1 -4035.653,E2 -4035.653} C_VEL
LIN {X 0,Y 538.593,Z 659.748,A -85,B 0,C 180,E1 -4036.8,E2 -4036.8} C_VEL
LIN {X 0,Y 538.283,Z 669.389,A -85,B 0,C 180,E1 -4037.942,E2 -4037.942} C_VEL
LIN {X 0,Y 538.068,Z 678.854,A -85,B 0,C 180,E1 -4039.273,E2 -4039.273} C_VEL
LIN {X 0,Y 537.824,Z 686.735,A -85,B 0,C 180,E1 -4040.599,E2 -4040.599} C_VEL
LIN {X 0,Y 537.699,Z 694.09,A -85,B 0,C 180,E1 -4042.112,E2 -4042.112} C_VEL
LIN {X 0,Y 537.626,Z 699.391,A -85,B 0,C 180,E1 -4043.459,E2 -4043.459} C_VEL
LIN {X 0,Y 537.574,Z 703.386,A -85,B 0,C 180,E1 -4044.749,E2 -4044.749} C_VEL
LIN {X 0,Y 537.562,Z 706.888,A -85,B 0,C 180,E1 -4046.252,E2 -4046.252} C_VEL
LIN {X 0,Y 537.487,Z 709.19,A -85,B 0,C 180,E1 -4047.752,E2 -4047.752} C_VEL
LIN {X 0,Y 537.438,Z 710.348,A -85,B 0,C 180,E1 -4049.251,E2 -4049.251} C_VEL
LIN {X 0,Y 537.438,Z 710.347,A -85,B 0,C 180,E1 -4050.749,E2 -4050.749} C_VEL
LIN {X 0,Y 537.487,Z 709.186,A -85,B 0,C 180,E1 -4052.248,E2 -4052.248} C_VEL
LIN {X 0,Y 537.562,Z 706.883,A -85,B 0,C 180,E1 -4053.748,E2 -4053.748} C_VEL
LIN {X 0,Y 537.574,Z 703.386,A -85,B 0,C 180,E1 -4055.251,E2 -4055.251} C_VEL
LIN {X 0,Y 537.618,Z 698.609,A -85,B 0,C 180,E1 -4056.757,E2 -4056.757} C_VEL
LIN {X 0,Y 537.734,Z 692.42,A -85,B 0,C 180,E1 -4058.266,E2 -4058.266} C_VEL
LIN {X 0,Y 537.859,Z 684.642,A -85,B 0,C 180,E1 -4059.78,E2 -4059.78} C_VEL
LIN {X 0,Y 538.101,Z 676.366,A -85,B 0,C 180,E1 -4061.107,E2 -4061.107} C_VEL
LIN {X 0,Y 538.358,Z 666.39,A -85,B 0,C 180,E1 -4062.439,E2 -4062.439} C_VEL
LIN {X 0,Y 538.662,Z 656.182,A -85,B 0,C 180,E1 -4063.583,E2 -4063.583} C_VEL
LIN {X 0,Y 539.03,Z 644.016,A -85,B 0,C 180,E1 -4064.729,E2 -4064.729} C_VEL
LIN {X 0,Y 539.468,Z 631.822,A -85,B 0,C 180,E1 -4065.682,E2 -4065.682} C_VEL
LIN {X 0,Y 539.826,Z 618.492,A -85,B 0,C 180,E1 -4066.546,E2 -4066.546} C_VEL
LIN {X 0,Y 540.165,Z 604.596,A -85,B 0,C 180,E1 -4067.266,E2 -4067.266} C_VEL
LIN {X 0,Y 540.497,Z 590.347,A -85,B 0,C 180,E1 -4067.841,E2 -4067.841} C_VEL
LIN {X 0,Y 540.799,Z 575.063,A -85,B 0,C 180,E1 -4068.297,E2 -4068.297} C_VEL
LIN {X 0,Y 540.943,Z 560.547,A -85,B 0,C 180,E1 -4068.588,E2 -4068.588} C_VEL
LIN {X 0,Y 541.703,Z 408.459,A -85,B 0,C 180,E1 -4070.652,E2 -4070.652} C_VEL
LIN {X 0,Y 539.871,Z 397.936,A -85,B 0,C 180,E1 -4070.889,E2 -4070.889} C_VEL
LIN {X 0,Y 540.528,Z 370.043,A -85,B 0,C 180,E1 -4073.946,E2 -4073.946} C_VEL
LIN {X 0,Y 541.06,Z 349.974,A -85,B 0,C 180,E1 -4076.209,E2 -4076.209} C_VEL
LIN {X 0,Y 538.098,Z 338.269,A -85,B 0,C 180,E1 -4077.772,E2 -4077.772} C_VEL
LIN {X 0,Y 538.022,Z 338.095,A -85,B 0,C 180,E1 -4080.627,E2 -4080.627} C_VEL
LIN {X 0,Y 538.047,Z 338.09,A -85,B 0,C 180,E1 -4083.283,E2 -4083.283} C_VEL
LIN {X 0,Y 538.002,Z 338.092,A -85,B 0,C 180,E1 -4086.004,E2 -4086.004} C_VEL
LIN {X 0,Y 538.014,Z 338.097,A -85,B 0,C 180,E1 -4088.831,E2 -4088.831} C_VEL
LIN {X 0,Y 538.031,Z 338.087,A -85,B 0,C 180,E1 -4091.773,E2 -4091.773} C_VEL
LIN {X 0,Y 538.007,Z 338.096,A -85,B 0,C 180,E1 -4094.862,E2 -4094.862} C_VEL
LIN {X 0,Y 538.001,Z 338.093,A -85,B 0,C 180,E1 -4097.212,E2 -4097.212} C_VEL
LIN {X 0,Y 538.022,Z 338.094,A -85,B 0,C 180,E1 -4100.203,E2 -4100.203} C_VEL
LIN {X 0,Y 538.019,Z 338.091,A -85,B 0,C 180,E1 -4103.067,E2 -4103.067} C_VEL
LIN {X 0,Y 538.007,Z 338.094,A -85,B 0,C 180,E1 -4105.826,E2 -4105.826} C_VEL
LIN {X 0,Y 538.008,Z 338.096,A -85,B 0,C 180,E1 -4108.499,E2 -4108.499} C_VEL
LIN {X 0,Y 537.985,Z 338.097,A -85,B 0,C 180,E1 -4111.096,E2 -4111.096} C_VEL
LIN {X 0,Y 538.021,Z 338.27,A -85,B 0,C 180,E1 -4113.739,E2 -4113.739} C_VEL
LIN {X 0,Y 540.319,Z 348.855,A -85,B 0,C 180,E1 -4115.403,E2 -4115.403} C_VEL
LIN {X 0,Y 539.721,Z 369.01,A -85,B 0,C 180,E1 -4118.216,E2 -4118.216} C_VEL
LIN {X 0,Y 539.174,Z 392.026,A -85,B 0,C 180,E1 -4121.376,E2 -4121.376} C_VEL
LIN {X 0,Y 539.048,Z 397.659,A -85,B 0,C 180,E1 -4122.109,E2 -4122.109} C_VEL
LIN {X 0,Y 540.751,Z 408.026,A -85,B 0,C 180,E1 -4122.349,E2 -4122.349} C_VEL
LIN {X 0,Y 540.075,Z 535.469,A -85,B 0,C 180,E1 -4124.117,E2 -4124.117} C_VEL
LIN {X 0,Y 539.831,Z 549.78,A -85,B 0,C 180,E1 -4124.46,E2 -4124.46} C_VEL
LIN {X 0,Y 539.639,Z 563.619,A -85,B 0,C 180,E1 -4124.95,E2 -4124.95} C_VEL
LIN {X 0,Y 539.373,Z 576.76,A -85,B 0,C 180,E1 -4125.57,E2 -4125.57} C_VEL
LIN {X 0,Y 538.997,Z 589.473,A -85,B 0,C 180,E1 -4126.33,E2 -4126.33} C_VEL
LIN {X 0,Y 538.732,Z 600.907,A -85,B 0,C 180,E1 -4127.187,E2 -4127.187} C_VEL
LIN {X 0,Y 538.413,Z 612.474,A -85,B 0,C 180,E1 -4128.235,E2 -4128.235} C_VEL
LIN {X 0,Y 538.209,Z 621.888,A -85,B 0,C 180,E1 -4129.276,E2 -4129.276} C_VEL
LIN {X 0,Y 537.974,Z 630.603,A -85,B 0,C 180,E1 -4130.412,E2 -4130.412} C_VEL
LIN {X 0,Y 537.811,Z 638.807,A -85,B 0,C 180,E1 -4131.735,E2 -4131.735} C_VEL
LIN {X 0,Y 537.661,Z 644.625,A -85,B 0,C 180,E1 -4132.867,E2 -4132.867} C_VEL
LIN {X 0,Y 537.656,Z 650.755,A -85,B 0,C 180,E1 -4134.374,E2 -4134.374} C_VEL
LIN {X 0,Y 537.55,Z 654.286,A -85,B 0,C 180,E1 -4135.501,E2 -4135.501} C_VEL
LIN {X 0,Y 537.547,Z 657.769,A -85,B 0,C 180,E1 -4137.002,E2 -4137.002} C_VEL
LIN {X 0,Y 537.45,Z 659.745,A -85,B 0,C 180,E1 -4138.501,E2 -4138.501} C_VEL
LIN {X 0,Y 537.441,Z 660.496,A -85,B 0,C 180,E1 -4140,E2 -4140} C_VEL
LIN {X 0,Y 537.447,Z 659.822,A -85,B 0,C 180,E1 -4141.499,E2 -4141.499} C_VEL
LIN {X 0,Y 537.546,Z 657.922,A -85,B 0,C 180,E1 -4142.998,E2 -4142.998} C_VEL
LIN {X 0,Y 537.55,Z 654.535,A -85,B 0,C 180,E1 -4144.499,E2 -4144.499} C_VEL
LIN {X 0,Y 537.655,Z 649.766,A -85,B 0,C 180,E1 -4146.003,E2 -4146.003} C_VEL
LIN {X 0,Y 537.662,Z 645.039,A -85,B 0,C 180,E1 -4147.133,E2 -4147.133} C_VEL
LIN {X 0,Y 537.823,Z 638.268,A -85,B 0,C 180,E1 -4148.454,E2 -4148.454} C_VEL
LIN {X 0,Y 537.948,Z 629.847,A -85,B 0,C 180,E1 -4149.778,E2 -4149.778} C_VEL
LIN {X 0,Y 538.216,Z 621.08,A -85,B 0,C 180,E1 -4150.914,E2 -4150.914} C_VEL
LIN {X 0,Y 538.451,Z 610.444,A -85,B 0,C 180,E1 -4152.054,E2 -4152.054} C_VEL
LIN {X 0,Y 538.765,Z 599.692,A -85,B 0,C 180,E1 -4153.004,E2 -4153.004} C_VEL
LIN {X 0,Y 539.041,Z 587.879,A -85,B 0,C 180,E1 -4153.861,E2 -4153.861} C_VEL
LIN {X 0,Y 539.408,Z 574.873,A -85,B 0,C 180,E1 -4154.622,E2 -4154.622} C_VEL
LIN {X 0,Y 539.712,Z 562.94,A -85,B 0,C 180,E1 -4155.167,E2 -4155.167} C_VEL
LIN {X 0,Y 539.886,Z 549.688,A -85,B 0,C 180,E1 -4155.632,E2 -4155.632} C_VEL
LIN {X 0,Y 540.076,Z 536.575,A -85,B 0,C 180,E1 -4155.956,E2 -4155.956} C_VEL
LIN {X 0,Y 540.399,Z 481.384,A -85,B 0,C 180,E1 -4156.723,E2 -4156.723} C_VEL
LIN {X 0,Y 540.62,Z 406.553,A -85,B 0,C 180,E1 -4157.75,E2 -4157.75} C_VEL
LIN {X 0,Y 538.993,Z 397.456,A -85,B 0,C 180,E1 -4157.966,E2 -4157.966} C_VEL
LIN {X 0,Y 539.417,Z 377.489,A -85,B 0,C 180,E1 -4160.655,E2 -4160.655} C_VEL
LIN {X 0,Y 538.889,Z 374.005,A -85,B 0,C 180,E1 -4161.159,E2 -4161.159} C_VEL
LIN {X 0,Y 533.593,Z 363.487,A -85,B 0,C 180,E1 -4162.87,E2 -4162.87} C_VEL
LIN {X 0,Y 533.099,Z 360.019,A -85,B 0,C 180,E1 -4163.384,E2 -4163.384} C_VEL
LIN {X 0,Y 533.366,Z 350.665,A -85,B 0,C 180,E1 -4164.703,E2 -4164.703} C_VEL
LIN {X 0,Y 531.919,Z 343.217,A -85,B 0,C 180,E1 -4165.85,E2 -4165.85} C_VEL
LIN {X 0,Y 530.973,Z 339.138,A -85,B 0,C 180,E1 -4166.533,E2 -4166.533} C_VEL
LIN {X 0,Y 530.918,Z 338.976,A -85,B 0,C 180,E1 -4169.327,E2 -4169.327} C_VEL
LIN {X 0,Y 530.951,Z 338.976,A -85,B 0,C 180,E1 -4172.097,E2 -4172.097} C_VEL
LIN {X 0,Y 530.952,Z 338.969,A -85,B 0,C 180,E1 -4174.848,E2 -4174.848} C_VEL
LIN {X 0,Y 530.925,Z 338.974,A -85,B 0,C 180,E1 -4177.511,E2 -4177.511} C_VEL
LIN {X 0,Y 530.907,Z 338.976,A -85,B 0,C 180,E1 -4180.44,E2 -4180.44} C_VEL
LIN {X 0,Y 530.92,Z 338.969,A -85,B 0,C 180,E1 -4183.499,E2 -4183.499} C_VEL
LIN {X 0,Y 530.961,Z 338.971,A -85,B 0,C 180,E1 -4185.624,E2 -4185.624} C_VEL
LIN {X 0,Y 530.907,Z 338.977,A -85,B 0,C 180,E1 -4188.556,E2 -4188.556} C_VEL
LIN {X 0,Y 530.929,Z 338.972,A -85,B 0,C 180,E1 -4191.527,E2 -4191.527} C_VEL
LIN {X 0,Y 530.925,Z 338.977,A -85,B 0,C 180,E1 -4194.378,E2 -4194.378} C_VEL
